LIN {X 0,Y 573.231,Z 369.083,A -85,B 0,C 180,E1 -2362.338,E2 -2362.338} C_VEL
LIN {X 0,Y 573.243,Z 369.081,A -85,B 0,C 180,E1 -2364.395,E2 -2364.395} C_VEL
LIN {X 0,Y 572.617,Z 369.161,A -85,B 0,C 180,E1 -2364.981,E2 -2364.981} C_VEL
LIN {X 0,Y 569.781,Z 369.515,A -85,B 0,C 180,E1 -2365.933,E2 -2365.933} C_VEL
LIN {X 0,Y 567.354,Z 369.816,A -85,B 0,C 180,E1 -2366.699,E2 -2366.699} C_VEL
LIN {X 0,Y 566.301,Z 369.946,A -85,B 0,C 180,E1 -2367.29,E2 -2367.29} C_VEL
LIN {X 0,Y 566.212,Z 369.956,A -85,B 0,C 180,E1 -2367.49,E2 -2367.49} C_VEL
LIN {X 0,Y 566.181,Z 369.961,A -85,B 0,C 180,E1 -2370.593,E2 -2370.593} C_VEL
LIN {X 0,Y 566.223,Z 369.955,A -85,B 0,C 180,E1 -2373.102,E2 -2373.102} C_VEL
LIN {X 0,Y 566.208,Z 369.958,A -85,B 0,C 180,E1 -2375.689,E2 -2375.689} C_VEL
LIN {X 0,Y 566.212,Z 369.957,A -85,B 0,C 180,E1 -2378.56,E2 -2378.56} C_VEL
LIN {X 0,Y 566.207,Z 369.958,A -85,B 0,C 180,E1 -2381.137,E2 -2381.137} C_VEL
LIN {X 0,Y 566.193,Z 369.96,A -85,B 0,C 180,E1 -2384.037,E2 -2384.037} C_VEL
LIN {X 0,Y 566.201,Z 369.96,A -85,B 0,C 180,E1 -2387.083,E2 -2387.083} C_VEL
LIN {X 0,Y 566.225,Z 369.955,A -85,B 0,C 180,E1 -2389.804,E2 -2389.804} C_VEL
LIN {X 0,Y 566.197,Z 369.96,A -85,B 0,C 180,E1 -2392.6,E2 -2392.6} C_VEL
LIN {X 0,Y 566.208,Z 369.957,A -85,B 0,C 180,E1 -2395.183,E2 -2395.183} C_VEL
LIN {X 0,Y 566.232,Z 369.955,A -85,B 0,C 180,E1 -2397.744,E2 -2397.744} C_VEL
LIN {X 0,Y 566.205,Z 369.959,A -85,B 0,C 180,E1 -2400.329,E2 -2400.329} C_VEL
LIN {X 0,Y 566.209,Z 369.958,A -85,B 0,C 180,E1 -2402.662,E2 -2402.662} C_VEL
LIN {X 0,Y 566.238,Z 369.953,A -85,B 0,C 180,E1 -2405.04,E2 -2405.04} C_VEL
LIN {X 0,Y 566.196,Z 369.96,A -85,B 0,C 180,E1 -2408.138,E2 -2408.138} C_VEL
LIN {X 0,Y 566.233,Z 369.954,A -85,B 0,C 180,E1 -2410.615,E2 -2410.615} C_VEL
LIN {X 0,Y 566.214,Z 369.958,A -85,B 0,C 180,E1 -2413.413,E2 -2413.413} C_VEL
LIN {X 0,Y 566.201,Z 369.958,A -85,B 0,C 180,E1 -2416.359,E2 -2416.359} C_VEL
LIN {X 0,Y 566.239,Z 369.953,A -85,B 0,C 180,E1 -2418.676,E2 -2418.676} C_VEL
LIN {X 0,Y 566.231,Z 369.956,A -85,B 0,C 180,E1 -2421.435,E2 -2421.435} C_VEL
LIN {X 0,Y 566.264,Z 369.951,A -85,B 0,C 180,E1 -2424.302,E2 -2424.302} C_VEL
LIN {X 0,Y 566.111,Z 369.972,A -85,B 0,C 180,E1 -2427.154,E2 -2427.154} C_VEL
LIN {X 0,Y 566.076,Z 369.978,A -85,B 0,C 180,E1 -2427.866,E2 -2427.866} C_VEL
LIN {X 0,Y 566.127,Z 372.153,A -85,B 0,C 180,E1 -2430,E2 -2430} C_VEL
LIN {X 0,Y 565.984,Z 374.62,A -85,B 0,C 180,E1 -2432.135,E2 -2432.135} C_VEL
LIN {X 0,Y 566.002,Z 377.796,A -85,B 0,C 180,E1 -2434.986,E2 -2434.986} C_VEL
LIN {X 0,Y 565.951,Z 381.039,A -85,B 0,C 180,E1 -2437.851,E2 -2437.851} C_VEL
LIN {X 0,Y 565.924,Z 384.456,A -85,B 0,C 180,E1 -2440.736,E2 -2440.736} C_VEL
LIN {X 0,Y 565.889,Z 388.157,A -85,B 0,C 180,E1 -2443.649,E2 -2443.649} C_VEL
LIN {X 0,Y 565.866,Z 391.969,A -85,B 0,C 180,E1 -2446.598,E2 -2446.598} C_VEL
LIN {X 0,Y 565.877,Z 395.756,A -85,B 0,C 180,E1 -2449.44,E2 -2449.44} C_VEL
LIN {X 0,Y 566.903,Z 403.162,A -85,B 0,C 180,E1 -2449.626,E2 -2449.626} C_VEL
LIN {X 0,Y 566.751,Z 416.361,A -85,B 0,C 180,E1 -2450.033,E2 -2450.033} C_VEL
LIN {X 0,Y 566.642,Z 427.451,A -85,B 0,C 180,E1 -2450.51,E2 -2450.51} C_VEL
LIN {X 0,Y 566.533,Z 439.685,A -85,B 0,C 180,E1 -2451.199,E2 -2451.199} C_VEL
LIN {X 0,Y 566.374,Z 450.264,A -85,B 0,C 180,E1 -2451.951,E2 -2451.951} C_VEL
LIN {X 0,Y 566.228,Z 460.09,A -85,B 0,C 180,E1 -2452.814,E2 -2452.814} C_VEL
LIN {X 0,Y 566.098,Z 469.138,A -85,B 0,C 180,E1 -2453.796,E2 -2453.796} C_VEL
LIN {X 0,Y 566.022,Z 476.522,A -85,B 0,C 180,E1 -2454.775,E2 -2454.775} C_VEL
LIN {X 0,Y 565.988,Z 483.713,A -85,B 0,C 180,E1 -2455.957,E2 -2455.957} C_VEL
LIN {X 0,Y 565.936,Z 488.503,A -85,B 0,C 180,E1 -2456.953,E2 -2456.953} C_VEL
LIN {X 0,Y 565.881,Z 492.991,A -85,B 0,C 180,E1 -2458.16,E2 -2458.16} C_VEL
LIN {X 0,Y 565.892,Z 495.248,A -85,B 0,C 180,E1 -2458.97,E2 -2458.97} C_VEL
LIN {X 0,Y 565.871,Z 497.003,A -85,B 0,C 180,E1 -2459.787,E2 -2459.787} C_VEL
LIN {X 0,Y 565.867,Z 498.577,A -85,B 0,C 180,E1 -2461.021,E2 -2461.021} C_VEL
LIN {X 0,Y 565.845,Z 498.934,A -85,B 0,C 180,E1 -2462.372,E2 -2462.372} C_VEL
LIN {X 0,Y 565.868,Z 497.946,A -85,B 0,C 180,E1 -2463.681,E2 -2463.681} C_VEL
LIN {X 0,Y 565.862,Z 495.687,A -85,B 0,C 180,E1 -2464.943,E2 -2464.943} C_VEL
LIN {X 0,Y 565.919,Z 492.176,A -85,B 0,C 180,E1 -2466.174,E2 -2466.174} C_VEL
LIN {X 0,Y 565.941,Z 486.955,A -85,B 0,C 180,E1 -2467.48,E2 -2467.48} C_VEL
LIN {X 0,Y 565.989,Z 480.61,A -85,B 0,C 180,E1 -2468.68,E2 -2468.68} C_VEL
LIN {X 0,Y 566.069,Z 474.047,A -85,B 0,C 180,E1 -2469.667,E2 -2469.667} C_VEL
LIN {X 0,Y 566.161,Z 464.892,A -85,B 0,C 180,E1 -2470.78,E2 -2470.78} C_VEL
LIN {X 0,Y 566.284,Z 455.077,A -85,B 0,C 180,E1 -2471.74,E2 -2471.74} C_VEL
LIN {X 0,Y 566.397,Z 444.775,A -85,B 0,C 180,E1 -2472.55,E2 -2472.55} C_VEL
LIN {X 0,Y 566.531,Z 433.437,A -85,B 0,C 180,E1 -2473.266,E2 -2473.266} C_VEL
LIN {X 0,Y 566.667,Z 421.184,A -85,B 0,C 180,E1 -2473.866,E2 -2473.866} C_VEL
LIN {X 0,Y 566.849,Z 408.099,A -85,B 0,C 180,E1 -2474.33,E2 -2474.33} C_VEL
LIN {X 0,Y 566.734,Z 401.219,A -85,B 0,C 180,E1 -2474.516,E2 -2474.516} C_VEL
LIN {X 0,Y 565.817,Z 395.661,A -85,B 0,C 180,E1 -2474.675,E2 -2474.675} C_VEL
LIN {X 0,Y 565.838,Z 391.468,A -85,B 0,C 180,E1 -2477.878,E2 -2477.878} C_VEL
LIN {X 0,Y 565.82,Z 387.838,A -85,B 0,C 180,E1 -2480.693,E2 -2480.693} C_VEL
LIN {X 0,Y 565.874,Z 383.867,A -85,B 0,C 180,E1 -2483.83,E2 -2483.83} C_VEL
LIN {X 0,Y 565.898,Z 381.098,A -85,B 0,C 180,E1 -2486.312,E2 -2486.312} C_VEL
LIN {X 0,Y 566,Z 378.247,A -85,B 0,C 180,E1 -2488.954,E2 -2488.954} C_VEL
LIN {X 0,Y 565.998,Z 374.957,A -85,B 0,C 180,E1 -2491.846,E2 -2491.846} C_VEL
LIN {X 0,Y 566.029,Z 372.197,A -85,B 0,C 180,E1 -2494.242,E2 -2494.242} C_VEL
LIN {X 0,Y 566.046,Z 370.404,A -85,B 0,C 180,E1 -2495.812,E2 -2495.812} C_VEL
LIN {X 0,Y 566.111,Z 369.973,A -85,B 0,C 180,E1 -2496.731,E2 -2496.731} C_VEL
LIN {X 0,Y 566.212,Z 369.957,A -85,B 0,C 180,E1 -2498.902,E2 -2498.902} C_VEL
LIN {X 0,Y 566.208,Z 369.958,A -85,B 0,C 180,E1 -2501.172,E2 -2501.172} C_VEL
LIN {X 0,Y 566.209,Z 369.96,A -85,B 0,C 180,E1 -2503.412,E2 -2503.412} C_VEL
LIN {X 0,Y 566.191,Z 369.959,A -85,B 0,C 180,E1 -2506.359,E2 -2506.359} C_VEL
LIN {X 0,Y 566.269,Z 369.949,A -85,B 0,C 180,E1 -2508.654,E2 -2508.654} C_VEL
LIN {X 0,Y 566.229,Z 369.954,A -85,B 0,C 180,E1 -2511.434,E2 -2511.434} C_VEL
LIN {X 0,Y 566.254,Z 369.954,A -85,B 0,C 180,E1 -2514.302,E2 -2514.302} C_VEL
LIN {X 0,Y 566.277,Z 369.951,A -85,B 0,C 180,E1 -2517.866,E2 -2517.866} C_VEL
LIN {X 0,Y 566.301,Z 369.945,A -85,B 0,C 180,E1 -2520.711,E2 -2520.711} C_VEL
LIN {X 0,Y 566.185,Z 369.96,A -85,B 0,C 180,E1 -2523.558,E2 -2523.558} C_VEL
LIN {X 0,Y 566.253,Z 369.951,A -85,B 0,C 180,E1 -2525.698,E2 -2525.698} C_VEL
LIN {X 0,Y 566.225,Z 369.955,A -85,B 0,C 180,E1 -2528.566,E2 -2528.566} C_VEL
LIN {X 0,Y 566.245,Z 369.953,A -85,B 0,C 180,E1 -2531.454,E2 -2531.454} C_VEL
LIN {X 0,Y 566.227,Z 369.954,A -85,B 0,C 180,E1 -2534.507,E2 -2534.507} C_VEL
LIN {X 0,Y 566.199,Z 369.961,A -85,B 0,C 180,E1 -2537.332,E2 -2537.332} C_VEL
LIN {X 0,Y 566.208,Z 369.956,A -85,B 0,C 180,E1 -2540.337,E2 -2540.337} C_VEL
LIN {X 0,Y 566.183,Z 369.963,A -85,B 0,C 180,E1 -2543.404,E2 -2543.404} C_VEL
LIN {X 0,Y 566.221,Z 369.959,A -85,B 0,C 180,E1 -2545.749,E2 -2545.749} C_VEL
LIN {X 0,Y 566.202,Z 369.961,A -85,B 0,C 180,E1 -2548.203,E2 -2548.203} C_VEL
LIN {X 0,Y 566.185,Z 369.96,A -85,B 0,C 180,E1 -2551.077,E2 -2551.077} C_VEL
LIN {X 0,Y 566.193,Z 369.959,A -85,B 0,C 180,E1 -2553.732,E2 -2553.732} C_VEL
LIN {X 0,Y 566.195,Z 369.962,A -85,B 0,C 180,E1 -2556.57,E2 -2556.57} C_VEL
LIN {X 0,Y 566.219,Z 369.958,A -85,B 0,C 180,E1 -2559.273,E2 -2559.273} C_VEL
LIN {X 0,Y 566.21,Z 369.956,A -85,B 0,C 180,E1 -2562.088,E2 -2562.088} C_VEL
LIN {X 0,Y 566.171,Z 369.964,A -85,B 0,C 180,E1 -2565.036,E2 -2565.036} C_VEL
LIN {X 0,Y 566.216,Z 369.957,A -85,B 0,C 180,E1 -2568.136,E2 -2568.136} C_VEL
LIN {X 0,Y 566.219,Z 369.957,A -85,B 0,C 180,E1 -2570.727,E2 -2570.727} C_VEL
LIN {X 0,Y 566.235,Z 369.971,A -85,B 0,C 180,E1 -2572.989,E2 -2572.989} C_VEL
LIN {X 0,Y 566.844,Z 373.918,A -85,B 0,C 180,E1 -2574.358,E2 -2574.358} C_VEL
LIN {X 0,Y 566.738,Z 381.862,A -85,B 0,C 180,E1 -2576.932,E2 -2576.932} C_VEL
LIN {X 0,Y 566.609,Z 389.805,A -85,B 0,C 180,E1 -2579.433,E2 -2579.433} C_VEL
LIN {X 0,Y 566.49,Z 399.072,A -85,B 0,C 180,E1 -2582.275,E2 -2582.275} C_VEL
LIN {X 0,Y 566.408,Z 408.339,A -85,B 0,C 180,E1 -2585.047,E2 -2585.047} C_VEL
LIN {X 0,Y 566.323,Z 418.93,A -85,B 0,C 180,E1 -2588.143,E2 -2588.143} C_VEL
LIN {X 0,Y 566.193,Z 429.521,A -85,B 0,C 180,E1 -2591.172,E2 -2591.172} C_VEL
LIN {X 0,Y 566.115,Z 440.112,A -85,B 0,C 180,E1 -2594.15,E2 -2594.15} C_VEL
LIN {X 0,Y 566.005,Z 450.703,A -85,B 0,C 180,E1 -2597.085,E2 -2597.085} C_VEL
LIN {X 0,Y 566.014,Z 451.53,A -85,B 0,C 180,E1 -2597.313,E2 -2597.313} C_VEL
LIN {X 0,Y 566.932,Z 458.375,A -85,B 0,C 180,E1 -2597.471,E2 -2597.471} C_VEL
LIN {X 0,Y 566.842,Z 470.499,A -85,B 0,C 180,E1 -2597.787,E2 -2597.787} C_VEL
LIN {X 0,Y 566.679,Z 482.321,A -85,B 0,C 180,E1 -2598.228,E2 -2598.228} C_VEL
LIN {X 0,Y 566.54,Z 494.84,A -85,B 0,C 180,E1 -2598.86,E2 -2598.86} C_VEL
LIN {X 0,Y 566.433,Z 505.479,A -85,B 0,C 180,E1 -2599.545,E2 -2599.545} C_VEL
LIN {X 0,Y 566.301,Z 515.647,A -85,B 0,C 180,E1 -2600.355,E2 -2600.355} C_VEL
LIN {X 0,Y 566.166,Z 524.787,A -85,B 0,C 180,E1 -2601.253,E2 -2601.253} C_VEL
LIN {X 0,Y 566.08,Z 533.69,A -85,B 0,C 180,E1 -2602.33,E2 -2602.33} C_VEL
LIN {X 0,Y 565.967,Z 540.955,A -85,B 0,C 180,E1 -2603.422,E2 -2603.422} C_VEL
LIN {X 0,Y 566.004,Z 545.68,A -85,B 0,C 180,E1 -2604.299,E2 -2604.299} C_VEL
LIN {X 0,Y 565.933,Z 550.371,A -85,B 0,C 180,E1 -2605.37,E2 -2605.37} C_VEL
LIN {X 0,Y 565.927,Z 553.956,A -85,B 0,C 180,E1 -2606.44,E2 -2606.44} C_VEL
LIN {X 0,Y 565.878,Z 555.808,A -85,B 0,C 180,E1 -2607.152,E2 -2607.152} C_VEL
LIN {X 0,Y 565.84,Z 557.2,A -85,B 0,C 180,E1 -2607.864,E2 -2607.864} C_VEL
LIN {X 0,Y 565.841,Z 558.784,A -85,B 0,C 180,E1 -2609.288,E2 -2609.288} C_VEL
LIN {X 0,Y 565.839,Z 559,A -85,B 0,C 180,E1 -2610,E2 -2610} C_VEL
LIN {X 0,Y 565.846,Z 558.186,A -85,B 0,C 180,E1 -2611.423,E2 -2611.423} C_VEL
LIN {X 0,Y 565.84,Z 557.201,A -85,B 0,C 180,E1 -2612.135,E2 -2612.135} C_VEL
LIN {X 0,Y 565.878,Z 555.81,A -85,B 0,C 180,E1 -2612.847,E2 -2612.847} C_VEL
LIN {X 0,Y 565.926,Z 552.897,A -85,B 0,C 180,E1 -2613.916,E2 -2613.916} C_VEL
LIN {X 0,Y 565.878,Z 548.951,A -85,B 0,C 180,E1 -2614.987,E2 -2614.987} C_VEL
LIN {X 0,Y 566.002,Z 543.868,A -85,B 0,C 180,E1 -2616.058,E2 -2616.058} C_VEL
LIN {X 0,Y 566.04,Z 537.472,A -85,B 0,C 180,E1 -2617.132,E2 -2617.132} C_VEL
LIN {X 0,Y 566.133,Z 529.481,A -85,B 0,C 180,E1 -2618.207,E2 -2618.207} C_VEL
LIN {X 0,Y 566.229,Z 521.34,A -85,B 0,C 180,E1 -2619.105,E2 -2619.105} C_VEL
LIN {X 0,Y 566.346,Z 511.407,A -85,B 0,C 180,E1 -2620.004,E2 -2620.004} C_VEL
LIN {X 0,Y 566.522,Z 500.32,A -85,B 0,C 180,E1 -2620.805,E2 -2620.805} C_VEL
LIN {X 0,Y 566.607,Z 487.959,A -85,B 0,C 180,E1 -2621.509,E2 -2621.509} C_VEL
LIN {X 0,Y 566.771,Z 475.779,A -85,B 0,C 180,E1 -2622.033,E2 -2622.033} C_VEL
LIN {X 0,Y 566.915,Z 463.282,A -85,B 0,C 180,E1 -2622.416,E2 -2622.416} C_VEL
LIN {X 0,Y 566.732,Z 456.109,A -85,B 0,C 180,E1 -2622.579,E2 -2622.579} C_VEL
LIN {X 0,Y 566.014,Z 451.532,A -85,B 0,C 180,E1 -2622.686,E2 -2622.686} C_VEL
LIN {X 0,Y 566.088,Z 441.437,A -85,B 0,C 180,E1 -2625.481,E2 -2625.481} C_VEL
LIN {X 0,Y 566.174,Z 430.846,A -85,B 0,C 180,E1 -2628.453,E2 -2628.453} C_VEL
LIN {X 0,Y 566.238,Z 421.579,A -85,B 0,C 180,E1 -2631.096,E2 -2631.096} C_VEL
LIN {X 0,Y 566.341,Z 412.312,A -85,B 0,C 180,E1 -2633.784,E2 -2633.784} C_VEL
LIN {X 0,Y 566.477,Z 403.045,A -85,B 0,C 180,E1 -2636.527,E2 -2636.527} C_VEL
LIN {X 0,Y 566.539,Z 393.778,A -85,B 0,C 180,E1 -2639.34,E2 -2639.34} C_VEL
LIN {X 0,Y 566.75,Z 384.511,A -85,B 0,C 180,E1 -2642.223,E2 -2642.223} C_VEL
LIN {X 0,Y 566.836,Z 376.568,A -85,B 0,C 180,E1 -2644.773,E2 -2644.773} C_VEL
LIN {X 0,Y 566.619,Z 372.042,A -85,B 0,C 180,E1 -2646.271,E2 -2646.271} C_VEL
LIN {X 0,Y 566.234,Z 369.955,A -85,B 0,C 180,E1 -2647.01,E2 -2647.01} C_VEL
LIN {X 0,Y 566.212,Z 369.959,A -85,B 0,C 180,E1 -2649.685,E2 -2649.685} C_VEL
LIN {X 0,Y 566.21,Z 369.958,A -85,B 0,C 180,E1 -2652.086,E2 -2652.086} C_VEL
LIN {X 0,Y 566.169,Z 369.965,A -85,B 0,C 180,E1 -2655.035,E2 -2655.035} C_VEL
LIN {X 0,Y 566.212,Z 369.957,A -85,B 0,C 180,E1 -2658.135,E2 -2658.135} C_VEL
LIN {X 0,Y 566.216,Z 369.959,A -85,B 0,C 180,E1 -2660.726,E2 -2660.726} C_VEL
LIN {X 0,Y 566.212,Z 369.958,A -85,B 0,C 180,E1 -2663.783,E2 -2663.783} C_VEL
LIN {X 0,Y 566.223,Z 369.958,A -85,B 0,C 180,E1 -2666.262,E2 -2666.262} C_VEL
LIN {X 0,Y 566.192,Z 369.959,A -85,B 0,C 180,E1 -2668.921,E2 -2668.921} C_VEL
LIN {X 0,Y 566.22,Z 369.957,A -85,B 0,C 180,E1 -2671.858,E2 -2671.858} C_VEL
LIN {X 0,Y 566.216,Z 369.957,A -85,B 0,C 180,E1 -2674.251,E2 -2674.251} C_VEL
LIN {X 0,Y 566.183,Z 369.96,A -85,B 0,C 180,E1 -2676.713,E2 -2676.713} C_VEL
LIN {X 0,Y 566.212,Z 369.957,A -85,B 0,C 180,E1 -2679.663,E2 -2679.663} C_VEL
LIN {X 0,Y 566.197,Z 369.96,A -85,B 0,C 180,E1 -2682.668,E2 -2682.668} C_VEL
LIN {X 0,Y 566.224,Z 369.955,A -85,B 0,C 180,E1 -2685.627,E2 -2685.627} C_VEL
LIN {X 0,Y 566.266,Z 369.951,A -85,B 0,C 180,E1 -2688.654,E2 -2688.654} C_VEL
LIN {X 0,Y 566.24,Z 369.955,A -85,B 0,C 180,E1 -2691.435,E2 -2691.435} C_VEL
LIN {X 0,Y 566.25,Z 369.952,A -85,B 0,C 180,E1 -2694.302,E2 -2694.302} C_VEL
LIN {X 0,Y 566.272,Z 369.949,A -85,B 0,C 180,E1 -2697.866,E2 -2697.866} C_VEL
LIN {X 0,Y 566.302,Z 369.947,A -85,B 0,C 180,E1 -2700.711,E2 -2700.711} C_VEL
LIN {X 0,Y 566.27,Z 369.951,A -85,B 0,C 180,E1 -2702.846,E2 -2702.846} C_VEL
LIN {X 0,Y 566.254,Z 369.951,A -85,B 0,C 180,E1 -2705.698,E2 -2705.698} C_VEL
LIN {X 0,Y 566.241,Z 369.954,A -85,B 0,C 180,E1 -2708.566,E2 -2708.566} C_VEL
LIN {X 0,Y 566.242,Z 369.955,A -85,B 0,C 180,E1 -2711.454,E2 -2711.454} C_VEL
LIN {X 0,Y 566.225,Z 369.956,A -85,B 0,C 180,E1 -2714.507,E2 -2714.507} C_VEL
LIN {X 0,Y 566.195,Z 369.959,A -85,B 0,C 180,E1 -2717.332,E2 -2717.332} C_VEL
LIN {X 0,Y 566.213,Z 369.959,A -85,B 0,C 180,E1 -2720.337,E2 -2720.337} C_VEL
LIN {X 0,Y 566.182,Z 369.96,A -85,B 0,C 180,E1 -2723.404,E2 -2723.404} C_VEL
LIN {X 0,Y 566.217,Z 369.957,A -85,B 0,C 180,E1 -2725.749,E2 -2725.749} C_VEL
LIN {X 0,Y 566.212,Z 369.956,A -85,B 0,C 180,E1 -2727.49,E2 -2727.49} C_VEL
LIN {X 0,Y 565.531,Z 370.044,A -85,B 0,C 180,E1 -2728.084,E2 -2728.084} C_VEL
LIN {X 0,Y 562.659,Z 370.4,A -85,B 0,C 180,E1 -2729.048,E2 -2729.048} C_VEL
LIN {X 0,Y 560.245,Z 370.7,A -85,B 0,C 180,E1 -2729.823,E2 -2729.823} C_VEL
LIN {X 0,Y 559.218,Z 370.83,A -85,B 0,C 180,E1 -2730.422,E2 -2730.422} C_VEL
LIN {X 0,Y 559.138,Z 370.836,A -85,B 0,C 180,E1 -2730.624,E2 -2730.624} C_VEL
LIN {X 0,Y 559.172,Z 370.835,A -85,B 0,C 180,E1 -2733.575,E2 -2733.575} C_VEL
LIN {X 0,Y 559.185,Z 370.832,A -85,B 0,C 180,E1 -2736.452,E2 -2736.452} C_VEL
LIN {X 0,Y 559.174,Z 370.834,A -85,B 0,C 180,E1 -2738.934,E2 -2738.934} C_VEL
LIN {X 0,Y 559.187,Z 370.832,A -85,B 0,C 180,E1 -2741.768,E2 -2741.768} C_VEL
LIN {X 0,Y 559.135,Z 370.84,A -85,B 0,C 180,E1 -2744.74,E2 -2744.74} C_VEL
LIN {X 0,Y 559.174,Z 370.834,A -85,B 0,C 180,E1 -2747.863,E2 -2747.863} C_VEL
LIN {X 0,Y 559.183,Z 370.834,A -85,B 0,C 180,E1 -2750.136,E2 -2750.136} C_VEL
LIN {X 0,Y 559.143,Z 370.837,A -85,B 0,C 180,E1 -2752.893,E2 -2752.893} C_VEL
LIN {X 0,Y 559.165,Z 370.836,A -85,B 0,C 180,E1 -2756.052,E2 -2756.052} C_VEL
LIN {X 0,Y 559.163,Z 370.836,A -85,B 0,C 180,E1 -2758.982,E2 -2758.982} C_VEL
LIN {X 0,Y 559.169,Z 370.835,A -85,B 0,C 180,E1 -2761.62,E2 -2761.62} C_VEL
LIN {X 0,Y 559.184,Z 370.833,A -85,B 0,C 180,E1 -2763.904,E2 -2763.904} C_VEL
LIN {X 0,Y 559.159,Z 370.836,A -85,B 0,C 180,E1 -2766.568,E2 -2766.568} C_VEL
LIN {X 0,Y 559.177,Z 370.834,A -85,B 0,C 180,E1 -2769.396,E2 -2769.396} C_VEL
LIN {X 0,Y 559.144,Z 370.838,A -85,B 0,C 180,E1 -2771.686,E2 -2771.686} C_VEL
LIN {X 0,Y 559.166,Z 370.835,A -85,B 0,C 180,E1 -2773.948,E2 -2773.948} C_VEL
LIN {X 0,Y 559.176,Z 370.833,A -85,B 0,C 180,E1 -2776.185,E2 -2776.185} C_VEL
LIN {X 0,Y 559.199,Z 370.833,A -85,B 0,C 180,E1 -2779.134,E2 -2779.134} C_VEL
LIN {X 0,Y 559.204,Z 370.83,A -85,B 0,C 180,E1 -2782.054,E2 -2782.054} C_VEL
LIN {X 0,Y 559.254,Z 370.823,A -85,B 0,C 180,E1 -2784.954,E2 -2784.954} C_VEL
LIN {X 0,Y 559.042,Z 370.854,A -85,B 0,C 180,E1 -2787.839,E2 -2787.839} C_VEL
LIN {X 0,Y 559.027,Z 371.145,A -85,B 0,C 180,E1 -2788.559,E2 -2788.559} C_VEL
LIN {X 0,Y 559.008,Z 373.635,A -85,B 0,C 180,E1 -2790.721,E2 -2790.721} C_VEL
LIN {X 0,Y 558.909,Z 376.925,A -85,B 0,C 180,E1 -2793.605,E2 -2793.605} C_VEL
LIN {X 0,Y 558.901,Z 379.335,A -85,B 0,C 180,E1 -2795.774,E2 -2795.774} C_VEL
LIN {X 0,Y 558.871,Z 382.614,A -85,B 0,C 180,E1 -2798.679,E2 -2798.679} C_VEL
LIN {X 0,Y 558.834,Z 385.979,A -85,B 0,C 180,E1 -2801.608,E2 -2801.608} C_VEL
LIN {X 0,Y 558.809,Z 389.63,A -85,B 0,C 180,E1 -2804.568,E2 -2804.568} C_VEL
LIN {X 0,Y 558.751,Z 393.48,A -85,B 0,C 180,E1 -2807.57,E2 -2807.57} C_VEL
LIN {X 0,Y 558.771,Z 395.776,A -85,B 0,C 180,E1 -2809.277,E2 -2809.277} C_VEL
LIN {X 0,Y 559.969,Z 403.84,A -85,B 0,C 180,E1 -2809.487,E2 -2809.487} C_VEL
LIN {X 0,Y 559.836,Z 415.759,A -85,B 0,C 180,E1 -2809.86,E2 -2809.86} C_VEL
LIN {X 0,Y 559.658,Z 428.016,A -85,B 0,C 180,E1 -2810.394,E2 -2810.394} C_VEL
LIN {X 0,Y 559.54,Z 439.834,A -85,B 0,C 180,E1 -2811.072,E2 -2811.072} C_VEL
LIN {X 0,Y 559.36,Z 450.423,A -85,B 0,C 180,E1 -2811.835,E2 -2811.835} C_VEL
LIN {X 0,Y 559.205,Z 460.456,A -85,B 0,C 180,E1 -2812.734,E2 -2812.734} C_VEL
LIN {X 0,Y 559.036,Z 469.387,A -85,B 0,C 180,E1 -2813.721,E2 -2813.721} C_VEL
LIN {X 0,Y 558.966,Z 477.487,A -85,B 0,C 180,E1 -2814.825,E2 -2814.825} C_VEL
LIN {X 0,Y 558.909,Z 483.87,A -85,B 0,C 180,E1 -2815.91,E2 -2815.91} C_VEL
LIN {X 0,Y 558.848,Z 488.636,A -85,B 0,C 180,E1 -2816.919,E2 -2816.919} C_VEL
LIN {X 0,Y 558.792,Z 493.576,A -85,B 0,C 180,E1 -2818.309,E2 -2818.309} C_VEL
LIN {X 0,Y 558.772,Z 497.053,A -85,B 0,C 180,E1 -2819.789,E2 -2819.789} C_VEL
LIN {X 0,Y 558.763,Z 498.71,A -85,B 0,C 180,E1 -2821.208,E2 -2821.208} C_VEL
LIN {X 0,Y 558.76,Z 498.89,A -85,B 0,C 180,E1 -2822.571,E2 -2822.571} C_VEL
LIN {X 0,Y 558.771,Z 497.69,A -85,B 0,C 180,E1 -2823.888,E2 -2823.888} C_VEL
LIN {X 0,Y 558.782,Z 495.241,A -85,B 0,C 180,E1 -2825.161,E2 -2825.161} C_VEL
LIN {X 0,Y 558.814,Z 491.588,A -85,B 0,C 180,E1 -2826.399,E2 -2826.399} C_VEL
LIN {X 0,Y 558.875,Z 486.709,A -85,B 0,C 180,E1 -2827.604,E2 -2827.604} C_VEL
LIN {X 0,Y 558.907,Z 480.552,A -85,B 0,C 180,E1 -2828.774,E2 -2828.774} C_VEL
LIN {X 0,Y 559.023,Z 472.853,A -85,B 0,C 180,E1 -2829.924,E2 -2829.924} C_VEL
LIN {X 0,Y 559.112,Z 464.514,A -85,B 0,C 180,E1 -2830.933,E2 -2830.933} C_VEL
LIN {X 0,Y 559.271,Z 455.125,A -85,B 0,C 180,E1 -2831.859,E2 -2831.859} C_VEL
LIN {X 0,Y 559.411,Z 444.27,A -85,B 0,C 180,E1 -2832.719,E2 -2832.719} C_VEL
LIN {X 0,Y 559.54,Z 432.266,A -85,B 0,C 180,E1 -2833.475,E2 -2833.475} C_VEL
LIN {X 0,Y 559.729,Z 420.751,A -85,B 0,C 180,E1 -2834.032,E2 -2834.032} C_VEL
LIN {X 0,Y 559.895,Z 407.507,A -85,B 0,C 180,E1 -2834.503,E2 -2834.503} C_VEL
LIN {X 0,Y 559.707,Z 401.571,A -85,B 0,C 180,E1 -2834.666,E2 -2834.666} C_VEL
LIN {X 0,Y 558.722,Z 395.672,A -85,B 0,C 180,E1 -2834.83,E2 -2834.83} C_VEL
LIN {X 0,Y 558.742,Z 391.69,A -85,B 0,C 180,E1 -2837.911,E2 -2837.911} C_VEL
LIN {X 0,Y 558.76,Z 388.889,A -85,B 0,C 180,E1 -2840.106,E2 -2840.106} C_VEL
LIN {X 0,Y 558.756,Z 385.618,A -85,B 0,C 180,E1 -2842.861,E2 -2842.861} C_VEL
LIN {X 0,Y 558.832,Z 382.587,A -85,B 0,C 180,E1 -2845.533,E2 -2845.533} C_VEL
LIN {X 0,Y 558.898,Z 379.772,A -85,B 0,C 180,E1 -2848.12,E2 -2848.12} C_VEL
LIN {X 0,Y 558.925,Z 376.983,A -85,B 0,C 180,E1 -2850.633,E2 -2850.633} C_VEL
LIN {X 0,Y 558.935,Z 374.024,A -85,B 0,C 180,E1 -2853.219,E2 -2853.219} C_VEL
LIN {X 0,Y 558.979,Z 371.475,A -85,B 0,C 180,E1 -2855.486,E2 -2855.486} C_VEL
LIN {X 0,Y 559.052,Z 370.852,A -85,B 0,C 180,E1 -2856.59,E2 -2856.59} C_VEL
LIN {X 0,Y 559.181,Z 370.833,A -85,B 0,C 180,E1 -2859.395,E2 -2859.395} C_VEL
LIN {X 0,Y 559.149,Z 370.836,A -85,B 0,C 180,E1 -2861.686,E2 -2861.686} C_VEL
LIN {X 0,Y 559.161,Z 370.834,A -85,B 0,C 180,E1 -2863.948,E2 -2863.948} C_VEL
LIN {X 0,Y 559.165,Z 370.834,A -85,B 0,C 180,E1 -2866.184,E2 -2866.184} C_VEL
LIN {X 0,Y 559.203,Z 370.83,A -85,B 0,C 180,E1 -2869.134,E2 -2869.134} C_VEL
LIN {X 0,Y 559.199,Z 370.831,A -85,B 0,C 180,E1 -2872.053,E2 -2872.053} C_VEL
LIN {X 0,Y 559.254,Z 370.822,A -85,B 0,C 180,E1 -2874.953,E2 -2874.953} C_VEL
LIN {X 0,Y 559.248,Z 370.826,A -85,B 0,C 180,E1 -2877.839,E2 -2877.839} C_VEL
LIN {X 0,Y 559.271,Z 370.821,A -85,B 0,C 180,E1 -2880.72,E2 -2880.72} C_VEL
LIN {X 0,Y 559.235,Z 370.827,A -85,B 0,C 180,E1 -2882.881,E2 -2882.881} C_VEL
LIN {X 0,Y 559.222,Z 370.827,A -85,B 0,C 180,E1 -2885.77,E2 -2885.77} C_VEL
LIN {X 0,Y 559.184,Z 370.833,A -85,B 0,C 180,E1 -2888.674,E2 -2888.674} C_VEL
LIN {X 0,Y 559.203,Z 370.83,A -85,B 0,C 180,E1 -2891.6,E2 -2891.6} C_VEL
LIN {X 0,Y 559.193,Z 370.831,A -85,B 0,C 180,E1 -2894.596,E2 -2894.596} C_VEL
LIN {X 0,Y 559.158,Z 370.836,A -85,B 0,C 180,E1 -2897.557,E2 -2897.557} C_VEL
LIN {X 0,Y 559.166,Z 370.836,A -85,B 0,C 180,E1 -2899.838,E2 -2899.838} C_VEL
LIN {X 0,Y 559.136,Z 370.841,A -85,B 0,C 180,E1 -2902.153,E2 -2902.153} C_VEL
LIN {X 0,Y 559.174,Z 370.833,A -85,B 0,C 180,E1 -2905.188,E2 -2905.188} C_VEL
LIN {X 0,Y 559.19,Z 370.831,A -85,B 0,C 180,E1 -2907.712,E2 -2907.712} C_VEL
LIN {X 0,Y 559.148,Z 370.837,A -85,B 0,C 180,E1 -2910.183,E2 -2910.183} C_VEL
LIN {X 0,Y 559.148,Z 370.837,A -85,B 0,C 180,E1 -2912.716,E2 -2912.716} C_VEL
LIN {X 0,Y 559.125,Z 370.842,A -85,B 0,C 180,E1 -2915.324,E2 -2915.324} C_VEL
LIN {X 0,Y 559.132,Z 370.841,A -85,B 0,C 180,E1 -2918.018,E2 -2918.018} C_VEL
LIN {X 0,Y 559.174,Z 370.833,A -85,B 0,C 180,E1 -2920.811,E2 -2920.811} C_VEL
LIN {X 0,Y 559.138,Z 370.839,A -85,B 0,C 180,E1 -2923.734,E2 -2923.734} C_VEL
LIN {X 0,Y 559.144,Z 370.838,A -85,B 0,C 180,E1 -2926.804,E2 -2926.804} C_VEL
LIN {X 0,Y 559.175,Z 370.835,A -85,B 0,C 180,E1 -2929.19,E2 -2929.19} C_VEL
LIN {X 0,Y 559.131,Z 370.84,A -85,B 0,C 180,E1 -2931.983,E2 -2931.983} C_VEL
LIN {X 0,Y 559.212,Z 371.017,A -85,B 0,C 180,E1 -2932.8,E2 -2932.8} C_VEL
LIN {X 0,Y 559.884,Z 375.26,A -85,B 0,C 180,E1 -2934.29,E2 -2934.29} C_VEL
LIN {X 0,Y 559.857,Z 381.862,A -85,B 0,C 180,E1 -2936.473,E2 -2936.473} C_VEL
LIN {X 0,Y 559.656,Z 389.805,A -85,B 0,C 180,E1 -2939.012,E2 -2939.012} C_VEL
LIN {X 0,Y 559.542,Z 399.159,A -85,B 0,C 180,E1 -2941.927,E2 -2941.927} C_VEL
LIN {X 0,Y 559.398,Z 408.516,A -85,B 0,C 180,E1 -2944.766,E2 -2944.766} C_VEL
LIN {X 0,Y 559.291,Z 418.93,A -85,B 0,C 180,E1 -2947.854,E2 -2947.854} C_VEL
LIN {X 0,Y 559.149,Z 429.521,A -85,B 0,C 180,E1 -2950.926,E2 -2950.926} C_VEL
LIN {X 0,Y 559.057,Z 438.788,A -85,B 0,C 180,E1 -2953.57,E2 -2953.57} C_VEL
LIN {X 0,Y 558.963,Z 449.379,A -85,B 0,C 180,E1 -2956.55,E2 -2956.55} C_VEL
LIN {X 0,Y 558.94,Z 451.53,A -85,B 0,C 180,E1 -2957.15,E2 -2957.15} C_VEL
LIN {X 0,Y 560.02,Z 459.514,A -85,B 0,C 180,E1 -2957.337,E2 -2957.337} C_VEL
LIN {X 0,Y 559.882,Z 471.879,A -85,B 0,C 180,E1 -2957.679,E2 -2957.679} C_VEL
LIN {X 0,Y 559.717,Z 484.284,A -85,B 0,C 180,E1 -2958.171,E2 -2958.171} C_VEL
LIN {X 0,Y 559.557,Z 495.668,A -85,B 0,C 180,E1 -2958.768,E2 -2958.768} C_VEL
LIN {X 0,Y 559.428,Z 506.747,A -85,B 0,C 180,E1 -2959.504,E2 -2959.504} C_VEL
LIN {X 0,Y 559.244,Z 517.601,A -85,B 0,C 180,E1 -2960.415,E2 -2960.415} C_VEL
LIN {X 0,Y 559.127,Z 526.413,A -85,B 0,C 180,E1 -2961.325,E2 -2961.325} C_VEL
LIN {X 0,Y 558.996,Z 535,A -85,B 0,C 180,E1 -2962.414,E2 -2962.414} C_VEL
LIN {X 0,Y 558.885,Z 542.688,A -85,B 0,C 180,E1 -2963.649,E2 -2963.649} C_VEL
LIN {X 0,Y 558.869,Z 547.365,A -85,B 0,C 180,E1 -2964.588,E2 -2964.588} C_VEL
LIN {X 0,Y 558.869,Z 551.677,A -85,B 0,C 180,E1 -2965.673,E2 -2965.673} C_VEL
LIN {X 0,Y 558.836,Z 553.956,A -85,B 0,C 180,E1 -2966.395,E2 -2966.395} C_VEL
LIN {X 0,Y 558.799,Z 555.808,A -85,B 0,C 180,E1 -2967.116,E2 -2967.116} C_VEL
LIN {X 0,Y 558.746,Z 557.199,A -85,B 0,C 180,E1 -2967.837,E2 -2967.837} C_VEL
LIN {X 0,Y 558.741,Z 558.784,A -85,B 0,C 180,E1 -2969.279,E2 -2969.279} C_VEL
LIN {X 0,Y 558.74,Z 559,A -85,B 0,C 180,E1 -2970,E2 -2970} C_VEL
LIN {X 0,Y 558.745,Z 558.186,A -85,B 0,C 180,E1 -2971.441,E2 -2971.441} C_VEL
LIN {X 0,Y 558.746,Z 557.201,A -85,B 0,C 180,E1 -2972.162,E2 -2972.162} C_VEL
LIN {X 0,Y 558.799,Z 555.81,A -85,B 0,C 180,E1 -2972.883,E2 -2972.883} C_VEL
LIN {X 0,Y 558.844,Z 552.897,A -85,B 0,C 180,E1 -2973.966,E2 -2973.966} C_VEL
LIN {X 0,Y 558.798,Z 548.95,A -85,B 0,C 180,E1 -2975.051,E2 -2975.051} C_VEL
LIN {X 0,Y 558.921,Z 543.868,A -85,B 0,C 180,E1 -2976.135,E2 -2976.135} C_VEL
LIN {X 0,Y 558.977,Z 537.472,A -85,B 0,C 180,E1 -2977.223,E2 -2977.223} C_VEL
LIN {X 0,Y 559.098,Z 529.481,A -85,B 0,C 180,E1 -2978.311,E2 -2978.311} C_VEL
LIN {X 0,Y 559.194,Z 521.34,A -85,B 0,C 180,E1 -2979.221,E2 -2979.221} C_VEL
LIN {X 0,Y 559.347,Z 511.407,A -85,B 0,C 180,E1 -2980.131,E2 -2980.131} C_VEL
LIN {X 0,Y 559.539,Z 500.416,A -85,B 0,C 180,E1 -2980.936,E2 -2980.936} C_VEL
LIN {X 0,Y 559.635,Z 488.831,A -85,B 0,C 180,E1 -2981.61,E2 -2981.61} C_VEL
LIN {X 0,Y 559.81,Z 476.999,A -85,B 0,C 180,E1 -2982.138,E2 -2982.138} C_VEL
LIN {X 0,Y 559.952,Z 464.195,A -85,B 0,C 180,E1 -2982.549,E2 -2982.549} C_VEL
LIN {X 0,Y 559.816,Z 456.967,A -85,B 0,C 180,E1 -2982.72,E2 -2982.72} C_VEL
LIN {X 0,Y 558.939,Z 451.532,A -85,B 0,C 180,E1 -2982.85,E2 -2982.85} C_VEL
LIN {X 0,Y 559.053,Z 441.437,A -85,B 0,C 180,E1 -2985.681,E2 -2985.681} C_VEL
LIN {X 0,Y 559.14,Z 430.846,A -85,B 0,C 180,E1 -2988.694,E2 -2988.694} C_VEL
LIN {X 0,Y 559.222,Z 420.92,A -85,B 0,C 180,E1 -2991.566,E2 -2991.566} C_VEL
LIN {X 0,Y 559.369,Z 410.988,A -85,B 0,C 180,E1 -2994.494,E2 -2994.494} C_VEL
LIN {X 0,Y 559.471,Z 401.721,A -85,B 0,C 180,E1 -2997.29,E2 -2997.29} C_VEL
LIN {X 0,Y 559.637,Z 392.454,A -85,B 0,C 180,E1 -3000.153,E2 -3000.153} C_VEL
LIN {X 0,Y 559.768,Z 384.329,A -85,B 0,C 180,E1 -3002.733,E2 -3002.733} C_VEL
LIN {X 0,Y 559.89,Z 376.376,A -85,B 0,C 180,E1 -3005.322,E2 -3005.322} C_VEL
LIN {X 0,Y 559.259,Z 371.193,A -85,B 0,C 180,E1 -3007.098,E2 -3007.098} C_VEL
LIN {X 0,Y 559.169,Z 370.837,A -85,B 0,C 180,E1 -3007.301,E2 -3007.301} C_VEL
LIN {X 0,Y 559.157,Z 370.836,A -85,B 0,C 180,E1 -3009.941,E2 -3009.941} C_VEL
LIN {X 0,Y 559.16,Z 370.837,A -85,B 0,C 180,E1 -3012.742,E2 -3012.742} C_VEL
LIN {X 0,Y 559.148,Z 370.837,A -85,B 0,C 180,E1 -3015.76,E2 -3015.76} C_VEL
LIN {X 0,Y 559.186,Z 370.833,A -85,B 0,C 180,E1 -3018.232,E2 -3018.232} C_VEL
LIN {X 0,Y 559.172,Z 370.834,A -85,B 0,C 180,E1 -3021.19,E2 -3021.19} C_VEL
LIN {X 0,Y 559.167,Z 370.836,A -85,B 0,C 180,E1 -3023.791,E2 -3023.791} C_VEL
LIN {X 0,Y 559.171,Z 370.835,A -85,B 0,C 180,E1 -3026.426,E2 -3026.426} C_VEL
LIN {X 0,Y 559.155,Z 370.836,A -85,B 0,C 180,E1 -3028.981,E2 -3028.981} C_VEL
LIN {X 0,Y 559.188,Z 370.831,A -85,B 0,C 180,E1 -3032.288,E2 -3032.288} C_VEL
LIN {X 0,Y 559.171,Z 370.835,A -85,B 0,C 180,E1 -3034.812,E2 -3034.812} C_VEL
LIN {X 0,Y 559.134,Z 370.837,A -85,B 0,C 180,E1 -3037.847,E2 -3037.847} C_VEL
LIN {X 0,Y 559.189,Z 370.833,A -85,B 0,C 180,E1 -3040.492,E2 -3040.492} C_VEL
LIN {X 0,Y 559.178,Z 370.833,A -85,B 0,C 180,E1 -3043.197,E2 -3043.197} C_VEL
LIN {X 0,Y 559.164,Z 370.837,A -85,B 0,C 180,E1 -3046.184,E2 -3046.184} C_VEL
LIN {X 0,Y 559.202,Z 370.831,A -85,B 0,C 180,E1 -3049.134,E2 -3049.134} C_VEL
LIN {X 0,Y 559.204,Z 370.83,A -85,B 0,C 180,E1 -3052.054,E2 -3052.054} C_VEL
LIN {X 0,Y 559.244,Z 370.827,A -85,B 0,C 180,E1 -3054.953,E2 -3054.953} C_VEL
LIN {X 0,Y 559.243,Z 370.824,A -85,B 0,C 180,E1 -3057.839,E2 -3057.839} C_VEL
LIN {X 0,Y 559.271,Z 370.822,A -85,B 0,C 180,E1 -3060.72,E2 -3060.72} C_VEL
LIN {X 0,Y 559.236,Z 370.827,A -85,B 0,C 180,E1 -3062.881,E2 -3062.881} C_VEL
LIN {X 0,Y 559.223,Z 370.827,A -85,B 0,C 180,E1 -3065.77,E2 -3065.77} C_VEL
LIN {X 0,Y 559.196,Z 370.831,A -85,B 0,C 180,E1 -3068.674,E2 -3068.674} C_VEL
LIN {X 0,Y 559.2,Z 370.832,A -85,B 0,C 180,E1 -3071.601,E2 -3071.601} C_VEL
LIN {X 0,Y 559.19,Z 370.832,A -85,B 0,C 180,E1 -3074.596,E2 -3074.596} C_VEL
LIN {X 0,Y 559.155,Z 370.835,A -85,B 0,C 180,E1 -3077.557,E2 -3077.557} C_VEL
LIN {X 0,Y 559.167,Z 370.834,A -85,B 0,C 180,E1 -3079.838,E2 -3079.838} C_VEL
LIN {X 0,Y 559.135,Z 370.838,A -85,B 0,C 180,E1 -3082.153,E2 -3082.153} C_VEL
LIN {X 0,Y 559.172,Z 370.833,A -85,B 0,C 180,E1 -3085.188,E2 -3085.188} C_VEL
LIN {X 0,Y 559.189,Z 370.831,A -85,B 0,C 180,E1 -3087.712,E2 -3087.712} C_VEL
LIN {X 0,Y 559.138,Z 370.836,A -85,B 0,C 180,E1 -3090.624,E2 -3090.624} C_VEL
LIN {X 0,Y 558.48,Z 370.921,A -85,B 0,C 180,E1 -3091.226,E2 -3091.226} C_VEL
LIN {X 0,Y 555.621,Z 371.276,A -85,B 0,C 180,E1 -3092.202,E2 -3092.202} C_VEL
LIN {X 0,Y 553.21,Z 371.576,A -85,B 0,C 180,E1 -3092.988,E2 -3092.988} C_VEL
LIN {X 0,Y 552.191,Z 371.704,A -85,B 0,C 180,E1 -3093.594,E2 -3093.594} C_VEL
LIN {X 0,Y 552.118,Z 371.711,A -85,B 0,C 180,E1 -3093.8,E2 -3093.8} C_VEL
LIN {X 0,Y 552.113,Z 371.714,A -85,B 0,C 180,E1 -3096.747,E2 -3096.747} C_VEL
LIN {X 0,Y 552.13,Z 371.711,A -85,B 0,C 180,E1 -3099.528,E2 -3099.528} C_VEL
LIN {X 0,Y 552.126,Z 371.713,A -85,B 0,C 180,E1 -3102.426,E2 -3102.426} C_VEL
LIN {X 0,Y 552.096,Z 371.715,A -85,B 0,C 180,E1 -3105.564,E2 -3105.564} C_VEL
LIN {X 0,Y 552.138,Z 371.71,A -85,B 0,C 180,E1 -3108.677,E2 -3108.677} C_VEL
LIN {X 0,Y 552.117,Z 371.714,A -85,B 0,C 180,E1 -3111.412,E2 -3111.412} C_VEL
LIN {X 0,Y 552.102,Z 371.715,A -85,B 0,C 180,E1 -3114.159,E2 -3114.159} C_VEL
LIN {X 0,Y 552.122,Z 371.714,A -85,B 0,C 180,E1 -3116.816,E2 -3116.816} C_VEL
LIN {X 0,Y 552.108,Z 371.715,A -85,B 0,C 180,E1 -3119.392,E2 -3119.392} C_VEL
LIN {X 0,Y 552.12,Z 371.712,A -85,B 0,C 180,E1 -3121.903,E2 -3121.903} C_VEL
LIN {X 0,Y 552.158,Z 371.709,A -85,B 0,C 180,E1 -3124.65,E2 -3124.65} C_VEL
LIN {X 0,Y 552.098,Z 371.715,A -85,B 0,C 180,E1 -3127.55,E2 -3127.55} C_VEL
LIN {X 0,Y 552.153,Z 371.707,A -85,B 0,C 180,E1 -3130.675,E2 -3130.675} C_VEL
LIN {X 0,Y 552.117,Z 371.714,A -85,B 0,C 180,E1 -3133.738,E2 -3133.738} C_VEL
LIN {X 0,Y 552.14,Z 371.71,A -85,B 0,C 180,E1 -3136.005,E2 -3136.005} C_VEL
LIN {X 0,Y 552.166,Z 371.708,A -85,B 0,C 180,E1 -3138.994,E2 -3138.994} C_VEL
LIN {X 0,Y 552.159,Z 371.708,A -85,B 0,C 180,E1 -3141.952,E2 -3141.952} C_VEL
LIN {X 0,Y 552.23,Z 371.699,A -85,B 0,C 180,E1 -3144.889,E2 -3144.889} C_VEL
LIN {X 0,Y 552.008,Z 371.73,A -85,B 0,C 180,E1 -3147.811,E2 -3147.811} C_VEL
LIN {X 0,Y 551.977,Z 371.78,A -85,B 0,C 180,E1 -3148.541,E2 -3148.541} C_VEL
LIN {X 0,Y 551.95,Z 374.273,A -85,B 0,C 180,E1 -3150.73,E2 -3150.73} C_VEL
LIN {X 0,Y 551.846,Z 378.416,A -85,B 0,C 180,E1 -3154.382,E2 -3154.382} C_VEL
LIN {X 0,Y 551.834,Z 381.697,A -85,B 0,C 180,E1 -3157.317,E2 -3157.317} C_VEL
LIN {X 0,Y 551.789,Z 385.06,A -85,B 0,C 180,E1 -3160.272,E2 -3160.272} C_VEL
LIN {X 0,Y 551.732,Z 387.581,A -85,B 0,C 180,E1 -3162.506,E2 -3162.506} C_VEL
LIN {X 0,Y 551.728,Z 390.161,A -85,B 0,C 180,E1 -3164.759,E2 -3164.759} C_VEL
LIN {X 0,Y 551.665,Z 394.02,A -85,B 0,C 180,E1 -3167.803,E2 -3167.803} C_VEL
LIN {X 0,Y 551.682,Z 395.68,A -85,B 0,C 180,E1 -3169.101,E2 -3169.101} C_VEL
LIN {X 0,Y 553.018,Z 405.082,A -85,B 0,C 180,E1 -3169.358,E2 -3169.358} C_VEL
LIN {X 0,Y 552.845,Z 417.531,A -85,B 0,C 180,E1 -3169.774,E2 -3169.774} C_VEL
LIN {X 0,Y 552.629,Z 430.478,A -85,B 0,C 180,E1 -3170.373,E2 -3170.373} C_VEL
LIN {X 0,Y 552.556,Z 441.76,A -85,B 0,C 180,E1 -3171.058,E2 -3171.058} C_VEL
LIN {X 0,Y 552.339,Z 451.982,A -85,B 0,C 180,E1 -3171.834,E2 -3171.834} C_VEL
LIN {X 0,Y 552.179,Z 460.742,A -85,B 0,C 180,E1 -3172.644,E2 -3172.644} C_VEL
LIN {X 0,Y 552.007,Z 468.893,A -85,B 0,C 180,E1 -3173.553,E2 -3173.553} C_VEL
LIN {X 0,Y 551.919,Z 476.916,A -85,B 0,C 180,E1 -3174.647,E2 -3174.647} C_VEL
LIN {X 0,Y 551.82,Z 484.025,A -85,B 0,C 180,E1 -3175.862,E2 -3175.862} C_VEL
LIN {X 0,Y 551.752,Z 488.912,A -85,B 0,C 180,E1 -3176.92,E2 -3176.92} C_VEL
LIN {X 0,Y 551.711,Z 493.165,A -85,B 0,C 180,E1 -3178.12,E2 -3178.12} C_VEL
LIN {X 0,Y 551.685,Z 495.398,A -85,B 0,C 180,E1 -3178.952,E2 -3178.952} C_VEL
LIN {X 0,Y 551.691,Z 497.38,A -85,B 0,C 180,E1 -3179.973,E2 -3179.973} C_VEL
LIN {X 0,Y 551.652,Z 498.838,A -85,B 0,C 180,E1 -3181.397,E2 -3181.397} C_VEL
LIN {X 0,Y 551.675,Z 498.786,A -85,B 0,C 180,E1 -3182.775,E2 -3182.775} C_VEL
LIN {X 0,Y 551.664,Z 497.407,A -85,B 0,C 180,E1 -3184.098,E2 -3184.098} C_VEL
LIN {X 0,Y 551.71,Z 494.791,A -85,B 0,C 180,E1 -3185.385,E2 -3185.385} C_VEL
LIN {X 0,Y 551.762,Z 490.454,A -85,B 0,C 180,E1 -3186.773,E2 -3186.773} C_VEL
LIN {X 0,Y 551.781,Z 485.928,A -85,B 0,C 180,E1 -3187.843,E2 -3187.843} C_VEL
LIN {X 0,Y 551.848,Z 479.546,A -85,B 0,C 180,E1 -3189.026,E2 -3189.026} C_VEL
LIN {X 0,Y 552.005,Z 471.641,A -85,B 0,C 180,E1 -3190.19,E2 -3190.19} C_VEL
LIN {X 0,Y 552.117,Z 463.64,A -85,B 0,C 180,E1 -3191.145,E2 -3191.145} C_VEL
LIN {X 0,Y 552.274,Z 454.466,A -85,B 0,C 180,E1 -3192.042,E2 -3192.042} C_VEL
LIN {X 0,Y 552.423,Z 444.448,A -85,B 0,C 180,E1 -3192.843,E2 -3192.843} C_VEL
LIN {X 0,Y 552.564,Z 432.41,A -85,B 0,C 180,E1 -3193.613,E2 -3193.613} C_VEL
LIN {X 0,Y 552.779,Z 420.585,A -85,B 0,C 180,E1 -3194.192,E2 -3194.192} C_VEL
LIN {X 0,Y 552.972,Z 407.41,A -85,B 0,C 180,E1 -3194.664,E2 -3194.664} C_VEL
LIN {X 0,Y 552.798,Z 402.637,A -85,B 0,C 180,E1 -3194.799,E2 -3194.799} C_VEL
LIN {X 0,Y 551.635,Z 395.666,A -85,B 0,C 180,E1 -3195.001,E2 -3195.001} C_VEL
LIN {X 0,Y 551.64,Z 392.3,A -85,B 0,C 180,E1 -3197.639,E2 -3197.639} C_VEL
LIN {X 0,Y 551.649,Z 388.913,A -85,B 0,C 180,E1 -3200.431,E2 -3200.431} C_VEL
LIN {X 0,Y 551.709,Z 385.698,A -85,B 0,C 180,E1 -3203.371,E2 -3203.371} C_VEL
LIN {X 0,Y 551.784,Z 382.843,A -85,B 0,C 180,E1 -3205.915,E2 -3205.915} C_VEL
LIN {X 0,Y 551.862,Z 379.946,A -85,B 0,C 180,E1 -3208.565,E2 -3208.565} C_VEL
LIN {X 0,Y 551.859,Z 376.663,A -85,B 0,C 180,E1 -3211.487,E2 -3211.487} C_VEL
LIN {X 0,Y 551.92,Z 373.086,A -85,B 0,C 180,E1 -3214.699,E2 -3214.699} C_VEL
LIN {X 0,Y 551.912,Z 371.741,A -85,B 0,C 180,E1 -3215.953,E2 -3215.953} C_VEL
LIN {X 0,Y 552.12,Z 371.715,A -85,B 0,C 180,E1 -3218.337,E2 -3218.337} C_VEL
LIN {X 0,Y 552.152,Z 371.709,A -85,B 0,C 180,E1 -3220.674,E2 -3220.674} C_VEL
LIN {X 0,Y 552.111,Z 371.713,A -85,B 0,C 180,E1 -3223.737,E2 -3223.737} C_VEL
LIN {X 0,Y 552.129,Z 371.712,A -85,B 0,C 180,E1 -3226.004,E2 -3226.004} C_VEL
LIN {X 0,Y 552.171,Z 371.705,A -85,B 0,C 180,E1 -3228.993,E2 -3228.993} C_VEL
LIN {X 0,Y 552.153,Z 371.709,A -85,B 0,C 180,E1 -3231.951,E2 -3231.951} C_VEL
LIN {X 0,Y 552.228,Z 371.697,A -85,B 0,C 180,E1 -3234.889,E2 -3234.889} C_VEL
LIN {X 0,Y 552.219,Z 371.701,A -85,B 0,C 180,E1 -3237.812,E2 -3237.812} C_VEL
LIN {X 0,Y 552.241,Z 371.697,A -85,B 0,C 180,E1 -3240.729,E2 -3240.729} C_VEL
LIN {X 0,Y 552.201,Z 371.703,A -85,B 0,C 180,E1 -3242.918,E2 -3242.918} C_VEL
LIN {X 0,Y 552.192,Z 371.702,A -85,B 0,C 180,E1 -3245.844,E2 -3245.844} C_VEL
LIN {X 0,Y 552.155,Z 371.71,A -85,B 0,C 180,E1 -3248.786,E2 -3248.786} C_VEL
LIN {X 0,Y 552.158,Z 371.707,A -85,B 0,C 180,E1 -3251.751,E2 -3251.751} C_VEL
LIN {X 0,Y 552.13,Z 371.712,A -85,B 0,C 180,E1 -3254.749,E2 -3254.749} C_VEL
LIN {X 0,Y 552.11,Z 371.713,A -85,B 0,C 180,E1 -3257.789,E2 -3257.789} C_VEL
LIN {X 0,Y 552.125,Z 371.711,A -85,B 0,C 180,E1 -3260.101,E2 -3260.101} C_VEL
LIN {X 0,Y 552.09,Z 371.716,A -85,B 0,C 180,E1 -3262.451,E2 -3262.451} C_VEL
LIN {X 0,Y 552.152,Z 371.708,A -85,B 0,C 180,E1 -3265.351,E2 -3265.351} C_VEL
LIN {X 0,Y 552.122,Z 371.714,A -85,B 0,C 180,E1 -3268.098,E2 -3268.098} C_VEL
LIN {X 0,Y 552.097,Z 371.718,A -85,B 0,C 180,E1 -3270.61,E2 -3270.61} C_VEL
LIN {X 0,Y 552.102,Z 371.717,A -85,B 0,C 180,E1 -3273.187,E2 -3273.187} C_VEL
LIN {X 0,Y 552.082,Z 371.718,A -85,B 0,C 180,E1 -3275.844,E2 -3275.844} C_VEL
LIN {X 0,Y 552.123,Z 371.715,A -85,B 0,C 180,E1 -3279.062,E2 -3279.062} C_VEL
LIN {X 0,Y 552.137,Z 371.713,A -85,B 0,C 180,E1 -3281.445,E2 -3281.445} C_VEL
LIN {X 0,Y 552.092,Z 371.715,A -85,B 0,C 180,E1 -3284.532,E2 -3284.532} C_VEL
LIN {X 0,Y 552.129,Z 371.714,A -85,B 0,C 180,E1 -3287.585,E2 -3287.585} C_VEL
LIN {X 0,Y 552.132,Z 371.712,A -85,B 0,C 180,E1 -3290.474,E2 -3290.474} C_VEL
LIN {X 0,Y 552.129,Z 371.758,A -85,B 0,C 180,E1 -3292.512,E2 -3292.512} C_VEL
LIN {X 0,Y 552.947,Z 376.594,A -85,B 0,C 180,E1 -3294.221,E2 -3294.221} C_VEL
LIN {X 0,Y 552.85,Z 384.509,A -85,B 0,C 180,E1 -3296.864,E2 -3296.864} C_VEL
LIN {X 0,Y 552.656,Z 393.796,A -85,B 0,C 180,E1 -3299.853,E2 -3299.853} C_VEL
LIN {X 0,Y 552.47,Z 403.044,A -85,B 0,C 180,E1 -3302.745,E2 -3302.745} C_VEL
LIN {X 0,Y 552.362,Z 410.987,A -85,B 0,C 180,E1 -3305.174,E2 -3305.174} C_VEL
LIN {X 0,Y 552.21,Z 421.578,A -85,B 0,C 180,E1 -3308.341,E2 -3308.341} C_VEL
LIN {X 0,Y 552.09,Z 430.845,A -85,B 0,C 180,E1 -3311.058,E2 -3311.058} C_VEL
LIN {X 0,Y 551.995,Z 441.436,A -85,B 0,C 180,E1 -3314.113,E2 -3314.113} C_VEL
LIN {X 0,Y 551.889,Z 451.53,A -85,B 0,C 180,E1 -3316.983,E2 -3316.983} C_VEL
LIN {X 0,Y 553.1,Z 460.526,A -85,B 0,C 180,E1 -3317.199,E2 -3317.199} C_VEL
LIN {X 0,Y 552.923,Z 473.179,A -85,B 0,C 180,E1 -3317.568,E2 -3317.568} C_VEL
LIN {X 0,Y 552.756,Z 485.486,A -85,B 0,C 180,E1 -3318.076,E2 -3318.076} C_VEL
LIN {X 0,Y 552.584,Z 497.21,A -85,B 0,C 180,E1 -3318.716,E2 -3318.716} C_VEL
LIN {X 0,Y 552.432,Z 507.928,A -85,B 0,C 180,E1 -3319.463,E2 -3319.463} C_VEL
LIN {X 0,Y 552.233,Z 517.601,A -85,B 0,C 180,E1 -3320.292,E2 -3320.292} C_VEL
LIN {X 0,Y 552.079,Z 526.413,A -85,B 0,C 180,E1 -3321.213,E2 -3321.213} C_VEL
LIN {X 0,Y 551.949,Z 535,A -85,B 0,C 180,E1 -3322.317,E2 -3322.317} C_VEL
LIN {X 0,Y 551.823,Z 541.867,A -85,B 0,C 180,E1 -3323.418,E2 -3323.418} C_VEL
LIN {X 0,Y 551.804,Z 547.365,A -85,B 0,C 180,E1 -3324.519,E2 -3324.519} C_VEL
LIN {X 0,Y 551.764,Z 551.677,A -85,B 0,C 180,E1 -3325.617,E2 -3325.617} C_VEL
LIN {X 0,Y 551.75,Z 553.957,A -85,B 0,C 180,E1 -3326.348,E2 -3326.348} C_VEL
LIN {X 0,Y 551.723,Z 555.808,A -85,B 0,C 180,E1 -3327.079,E2 -3327.079} C_VEL
LIN {X 0,Y 551.657,Z 557.199,A -85,B 0,C 180,E1 -3327.81,E2 -3327.81} C_VEL
LIN {X 0,Y 551.641,Z 558.785,A -85,B 0,C 180,E1 -3329.27,E2 -3329.27} C_VEL
LIN {X 0,Y 551.64,Z 559,A -85,B 0,C 180,E1 -3330,E2 -3330} C_VEL
LIN {X 0,Y 551.645,Z 558.186,A -85,B 0,C 180,E1 -3331.46,E2 -3331.46} C_VEL
LIN {X 0,Y 551.657,Z 557.201,A -85,B 0,C 180,E1 -3332.19,E2 -3332.19} C_VEL
LIN {X 0,Y 551.723,Z 555.81,A -85,B 0,C 180,E1 -3332.92,E2 -3332.92} C_VEL
LIN {X 0,Y 551.764,Z 552.897,A -85,B 0,C 180,E1 -3334.017,E2 -3334.017} C_VEL
LIN {X 0,Y 551.723,Z 548.95,A -85,B 0,C 180,E1 -3335.115,E2 -3335.115} C_VEL
LIN {X 0,Y 551.803,Z 543.19,A -85,B 0,C 180,E1 -3336.341,E2 -3336.341} C_VEL
LIN {X 0,Y 551.926,Z 536.239,A -85,B 0,C 180,E1 -3337.499,E2 -3337.499} C_VEL
LIN {X 0,Y 552.082,Z 527.993,A -85,B 0,C 180,E1 -3338.602,E2 -3338.602} C_VEL
LIN {X 0,Y 552.201,Z 519.542,A -85,B 0,C 180,E1 -3339.523,E2 -3339.523} C_VEL
LIN {X 0,Y 552.405,Z 509.101,A -85,B 0,C 180,E1 -3340.445,E2 -3340.445} C_VEL
LIN {X 0,Y 552.564,Z 498.297,A -85,B 0,C 180,E1 -3341.214,E2 -3341.214} C_VEL
LIN {X 0,Y 552.7,Z 487.42,A -85,B 0,C 180,E1 -3341.832,E2 -3341.832} C_VEL
LIN {X 0,Y 552.878,Z 475.775,A -85,B 0,C 180,E1 -3342.34,E2 -3342.34} C_VEL
LIN {X 0,Y 553.068,Z 462.367,A -85,B 0,C 180,E1 -3342.755,E2 -3342.755} C_VEL
LIN {X 0,Y 552.894,Z 457.823,A -85,B 0,C 180,E1 -3342.864,E2 -3342.864} C_VEL
LIN {X 0,Y 551.889,Z 451.532,A -85,B 0,C 180,E1 -3343.017,E2 -3343.017} C_VEL
LIN {X 0,Y 551.994,Z 441.437,A -85,B 0,C 180,E1 -3345.886,E2 -3345.886} C_VEL
LIN {X 0,Y 552.089,Z 430.846,A -85,B 0,C 180,E1 -3348.941,E2 -3348.941} C_VEL
LIN {X 0,Y 552.252,Z 420.257,A -85,B 0,C 180,E1 -3352.049,E2 -3352.049} C_VEL
LIN {X 0,Y 552.361,Z 410.988,A -85,B 0,C 180,E1 -3354.826,E2 -3354.826} C_VEL
LIN {X 0,Y 552.504,Z 401.721,A -85,B 0,C 180,E1 -3357.663,E2 -3357.663} C_VEL
LIN {X 0,Y 552.664,Z 392.454,A -85,B 0,C 180,E1 -3360.574,E2 -3360.574} C_VEL
LIN {X 0,Y 552.848,Z 384.511,A -85,B 0,C 180,E1 -3363.135,E2 -3363.135} C_VEL
LIN {X 0,Y 552.92,Z 376.467,A -85,B 0,C 180,E1 -3365.78,E2 -3365.78} C_VEL
LIN {X 0,Y 552.101,Z 371.717,A -85,B 0,C 180,E1 -3367.518,E2 -3367.518} C_VEL
LIN {X 0,Y 552.106,Z 371.715,A -85,B 0,C 180,E1 -3370.48,E2 -3370.48} C_VEL
LIN {X 0,Y 552.102,Z 371.715,A -85,B 0,C 180,E1 -3373.482,E2 -3373.482} C_VEL
LIN {X 0,Y 552.101,Z 371.715,A -85,B 0,C 180,E1 -3376.575,E2 -3376.575} C_VEL
LIN {X 0,Y 552.136,Z 371.713,A -85,B 0,C 180,E1 -3379.521,E2 -3379.521} C_VEL
LIN {X 0,Y 552.088,Z 371.716,A -85,B 0,C 180,E1 -3382.336,E2 -3382.336} C_VEL
LIN {X 0,Y 552.125,Z 371.714,A -85,B 0,C 180,E1 -3385.054,E2 -3385.054} C_VEL
LIN {X 0,Y 552.121,Z 371.711,A -85,B 0,C 180,E1 -3387.682,E2 -3387.682} C_VEL
LIN {X 0,Y 552.105,Z 371.713,A -85,B 0,C 180,E1 -3390.235,E2 -3390.235} C_VEL
LIN {X 0,Y 552.14,Z 371.711,A -85,B 0,C 180,E1 -3392.997,E2 -3392.997} C_VEL
LIN {X 0,Y 552.105,Z 371.715,A -85,B 0,C 180,E1 -3395.161,E2 -3395.161} C_VEL
LIN {X 0,Y 552.088,Z 371.716,A -85,B 0,C 180,E1 -3397.549,E2 -3397.549} C_VEL
LIN {X 0,Y 552.141,Z 371.71,A -85,B 0,C 180,E1 -3400.373,E2 -3400.373} C_VEL
LIN {X 0,Y 552.15,Z 371.709,A -85,B 0,C 180,E1 -3402.977,E2 -3402.977} C_VEL
LIN {X 0,Y 552.127,Z 371.712,A -85,B 0,C 180,E1 -3406.004,E2 -3406.004} C_VEL
LIN {X 0,Y 552.169,Z 371.706,A -85,B 0,C 180,E1 -3408.994,E2 -3408.994} C_VEL
LIN {X 0,Y 552.157,Z 371.708,A -85,B 0,C 180,E1 -3411.952,E2 -3411.952} C_VEL
LIN {X 0,Y 552.219,Z 371.702,A -85,B 0,C 180,E1 -3414.889,E2 -3414.889} C_VEL
LIN {X 0,Y 552.214,Z 371.699,A -85,B 0,C 180,E1 -3417.812,E2 -3417.812} C_VEL
LIN {X 0,Y 552.24,Z 371.698,A -85,B 0,C 180,E1 -3420.729,E2 -3420.729} C_VEL
LIN {X 0,Y 552.202,Z 371.703,A -85,B 0,C 180,E1 -3422.918,E2 -3422.918} C_VEL
LIN {X 0,Y 552.193,Z 371.703,A -85,B 0,C 180,E1 -3425.844,E2 -3425.844} C_VEL
LIN {X 0,Y 552.164,Z 371.707,A -85,B 0,C 180,E1 -3428.786,E2 -3428.786} C_VEL
LIN {X 0,Y 552.155,Z 371.709,A -85,B 0,C 180,E1 -3431.751,E2 -3431.751} C_VEL
LIN {X 0,Y 552.127,Z 371.713,A -85,B 0,C 180,E1 -3434.749,E2 -3434.749} C_VEL
LIN {X 0,Y 552.107,Z 371.713,A -85,B 0,C 180,E1 -3437.789,E2 -3437.789} C_VEL
LIN {X 0,Y 552.127,Z 371.712,A -85,B 0,C 180,E1 -3440.102,E2 -3440.102} C_VEL
LIN {X 0,Y 552.089,Z 371.717,A -85,B 0,C 180,E1 -3442.451,E2 -3442.451} C_VEL
LIN {X 0,Y 552.149,Z 371.707,A -85,B 0,C 180,E1 -3445.352,E2 -3445.352} C_VEL
LIN {X 0,Y 552.121,Z 371.714,A -85,B 0,C 180,E1 -3448.098,E2 -3448.098} C_VEL
LIN {X 0,Y 552.1,Z 371.715,A -85,B 0,C 180,E1 -3450.62,E2 -3450.62} C_VEL
LIN {X 0,Y 552.123,Z 371.711,A -85,B 0,C 180,E1 -3453.186,E2 -3453.186} C_VEL
LIN {X 0,Y 552.118,Z 371.711,A -85,B 0,C 180,E1 -3453.8,E2 -3453.8} C_VEL
LIN {X 0,Y 551.484,Z 371.793,A -85,B 0,C 180,E1 -3454.408,E2 -3454.408} C_VEL
LIN {X 0,Y 548.662,Z 372.148,A -85,B 0,C 180,E1 -3455.397,E2 -3455.397} C_VEL
LIN {X 0,Y 546.238,Z 372.45,A -85,B 0,C 180,E1 -3456.192,E2 -3456.192} C_VEL
LIN {X 0,Y 545.166,Z 372.581,A -85,B 0,C 180,E1 -3456.806,E2 -3456.806} C_VEL
LIN {X 0,Y 545.064,Z 372.592,A -85,B 0,C 180,E1 -3457.014,E2 -3457.014} C_VEL
LIN {X 0,Y 545.088,Z 372.589,A -85,B 0,C 180,E1 -3460.141,E2 -3460.141} C_VEL
LIN {X 0,Y 545.074,Z 372.589,A -85,B 0,C 180,E1 -3463.107,E2 -3463.107} C_VEL
LIN {X 0,Y 545.055,Z 372.593,A -85,B 0,C 180,E1 -3466.226,E2 -3466.226} C_VEL
LIN {X 0,Y 545.095,Z 372.588,A -85,B 0,C 180,E1 -3468.888,E2 -3468.888} C_VEL
LIN {X 0,Y 545.051,Z 372.593,A -85,B 0,C 180,E1 -3471.764,E2 -3471.764} C_VEL
LIN {X 0,Y 545.052,Z 372.594,A -85,B 0,C 180,E1 -3474.534,E2 -3474.534} C_VEL
LIN {X 0,Y 545.081,Z 372.589,A -85,B 0,C 180,E1 -3477.213,E2 -3477.213} C_VEL
LIN {X 0,Y 545.067,Z 372.591,A -85,B 0,C 180,E1 -3479.812,E2 -3479.812} C_VEL
LIN {X 0,Y 545.089,Z 372.59,A -85,B 0,C 180,E1 -3482.345,E2 -3482.345} C_VEL
LIN {X 0,Y 545.119,Z 372.585,A -85,B 0,C 180,E1 -3484.821,E2 -3484.821} C_VEL
LIN {X 0,Y 545.046,Z 372.593,A -85,B 0,C 180,E1 -3487.243,E2 -3487.243} C_VEL
LIN {X 0,Y 545.119,Z 372.585,A -85,B 0,C 180,E1 -3490.415,E2 -3490.415} C_VEL
LIN {X 0,Y 545.068,Z 372.593,A -85,B 0,C 180,E1 -3493.522,E2 -3493.522} C_VEL
LIN {X 0,Y 545.099,Z 372.589,A -85,B 0,C 180,E1 -3495.821,E2 -3495.821} C_VEL
LIN {X 0,Y 545.122,Z 372.585,A -85,B 0,C 180,E1 -3498.85,E2 -3498.85} C_VEL
LIN {X 0,Y 545.13,Z 372.583,A -85,B 0,C 180,E1 -3501.847,E2 -3501.847} C_VEL
LIN {X 0,Y 545.206,Z 372.574,A -85,B 0,C 180,E1 -3504.823,E2 -3504.823} C_VEL
LIN {X 0,Y 544.974,Z 372.606,A -85,B 0,C 180,E1 -3507.783,E2 -3507.783} C_VEL
LIN {X 0,Y 544.953,Z 372.61,A -85,B 0,C 180,E1 -3508.522,E2 -3508.522} C_VEL
LIN {X 0,Y 544.969,Z 374.068,A -85,B 0,C 180,E1 -3510,E2 -3510} C_VEL
LIN {X 0,Y 544.722,Z 377.448,A -85,B 0,C 180,E1 -3512.958,E2 -3512.958} C_VEL
LIN {X 0,Y 544.806,Z 379.929,A -85,B 0,C 180,E1 -3515.181,E2 -3515.181} C_VEL
LIN {X 0,Y 544.767,Z 382.438,A -85,B 0,C 180,E1 -3517.412,E2 -3517.412} C_VEL
LIN {X 0,Y 544.735,Z 385.807,A -85,B 0,C 180,E1 -3520.406,E2 -3520.406} C_VEL
LIN {X 0,Y 544.616,Z 389.199,A -85,B 0,C 180,E1 -3523.431,E2 -3523.431} C_VEL
LIN {X 0,Y 544.594,Z 391.776,A -85,B 0,C 180,E1 -3525.724,E2 -3525.724} C_VEL
LIN {X 0,Y 544.559,Z 394.562,A -85,B 0,C 180,E1 -3528.043,E2 -3528.043} C_VEL
LIN {X 0,Y 544.598,Z 395.667,A -85,B 0,C 180,E1 -3528.919,E2 -3528.919} C_VEL
LIN {X 0,Y 546.094,Z 405.516,A -85,B 0,C 180,E1 -3529.207,E2 -3529.207} C_VEL
LIN {X 0,Y 545.891,Z 418.712,A -85,B 0,C 180,E1 -3529.664,E2 -3529.664} C_VEL
LIN {X 0,Y 545.671,Z 430.297,A -85,B 0,C 180,E1 -3530.213,E2 -3530.213} C_VEL
LIN {X 0,Y 545.562,Z 442.185,A -85,B 0,C 180,E1 -3530.945,E2 -3530.945} C_VEL
LIN {X 0,Y 545.333,Z 452.064,A -85,B 0,C 180,E1 -3531.709,E2 -3531.709} C_VEL
LIN {X 0,Y 545.147,Z 461.032,A -85,B 0,C 180,E1 -3532.553,E2 -3532.553} C_VEL
LIN {X 0,Y 544.93,Z 469.877,A -85,B 0,C 180,E1 -3533.566,E2 -3533.566} C_VEL
LIN {X 0,Y 544.862,Z 477.116,A -85,B 0,C 180,E1 -3534.581,E2 -3534.581} C_VEL
LIN {X 0,Y 544.774,Z 483.576,A -85,B 0,C 180,E1 -3535.693,E2 -3535.693} C_VEL
LIN {X 0,Y 544.663,Z 488.888,A -85,B 0,C 180,E1 -3536.847,E2 -3536.847} C_VEL
LIN {X 0,Y 544.615,Z 493.254,A -85,B 0,C 180,E1 -3538.1,E2 -3538.1} C_VEL
LIN {X 0,Y 544.593,Z 496.365,A -85,B 0,C 180,E1 -3539.366,E2 -3539.366} C_VEL
LIN {X 0,Y 544.596,Z 497.787,A -85,B 0,C 180,E1 -3540.218,E2 -3540.218} C_VEL
LIN {X 0,Y 544.544,Z 498.909,A -85,B 0,C 180,E1 -3541.59,E2 -3541.59} C_VEL
LIN {X 0,Y 544.574,Z 498.659,A -85,B 0,C 180,E1 -3542.98,E2 -3542.98} C_VEL
LIN {X 0,Y 544.575,Z 497.118,A -85,B 0,C 180,E1 -3544.314,E2 -3544.314} C_VEL
LIN {X 0,Y 544.612,Z 494.339,A -85,B 0,C 180,E1 -3545.61,E2 -3545.61} C_VEL
LIN {X 0,Y 544.668,Z 490.323,A -85,B 0,C 180,E1 -3546.869,E2 -3546.869} C_VEL
LIN {X 0,Y 544.732,Z 485.078,A -85,B 0,C 180,E1 -3548.093,E2 -3548.093} C_VEL
LIN {X 0,Y 544.825,Z 478.518,A -85,B 0,C 180,E1 -3549.288,E2 -3549.288} C_VEL
LIN {X 0,Y 544.973,Z 470.39,A -85,B 0,C 180,E1 -3550.459,E2 -3550.459} C_VEL
LIN {X 0,Y 545.14,Z 461.269,A -85,B 0,C 180,E1 -3551.513,E2 -3551.513} C_VEL
LIN {X 0,Y 545.292,Z 451.362,A -85,B 0,C 180,E1 -3552.443,E2 -3552.443} C_VEL
LIN {X 0,Y 545.484,Z 441.525,A -85,B 0,C 180,E1 -3553.192,E2 -3553.192} C_VEL
LIN {X 0,Y 545.674,Z 429.878,A -85,B 0,C 180,E1 -3553.899,E2 -3553.899} C_VEL
LIN {X 0,Y 545.916,Z 417.13,A -85,B 0,C 180,E1 -3554.492,E2 -3554.492} C_VEL
LIN {X 0,Y 546.029,Z 404.5,A -85,B 0,C 180,E1 -3554.912,E2 -3554.912} C_VEL
LIN {X 0,Y 544.548,Z 395.672,A -85,B 0,C 180,E1 -3555.168,E2 -3555.168} C_VEL
LIN {X 0,Y 544.563,Z 392.401,A -85,B 0,C 180,E1 -3557.848,E2 -3557.848} C_VEL
LIN {X 0,Y 544.577,Z 389.211,A -85,B 0,C 180,E1 -3560.775,E2 -3560.775} C_VEL
LIN {X 0,Y 544.635,Z 386.103,A -85,B 0,C 180,E1 -3563.588,E2 -3563.588} C_VEL
LIN {X 0,Y 544.706,Z 383.107,A -85,B 0,C 180,E1 -3566.303,E2 -3566.303} C_VEL
LIN {X 0,Y 544.783,Z 380.213,A -85,B 0,C 180,E1 -3568.934,E2 -3568.934} C_VEL
LIN {X 0,Y 544.818,Z 377.329,A -85,B 0,C 180,E1 -3571.491,E2 -3571.491} C_VEL
LIN {X 0,Y 544.875,Z 373.65,A -85,B 0,C 180,E1 -3574.808,E2 -3574.808} C_VEL
LIN {X 0,Y 544.845,Z 372.766,A -85,B 0,C 180,E1 -3575.621,E2 -3575.621} C_VEL
LIN {X 0,Y 545.057,Z 372.594,A -85,B 0,C 180,E1 -3578.18,E2 -3578.18} C_VEL
LIN {X 0,Y 545.116,Z 372.585,A -85,B 0,C 180,E1 -3580.415,E2 -3580.415} C_VEL
LIN {X 0,Y 545.068,Z 372.592,A -85,B 0,C 180,E1 -3583.521,E2 -3583.521} C_VEL
LIN {X 0,Y 545.088,Z 372.591,A -85,B 0,C 180,E1 -3585.82,E2 -3585.82} C_VEL
LIN {X 0,Y 545.126,Z 372.582,A -85,B 0,C 180,E1 -3588.849,E2 -3588.849} C_VEL
LIN {X 0,Y 545.124,Z 372.586,A -85,B 0,C 180,E1 -3591.847,E2 -3591.847} C_VEL
LIN {X 0,Y 545.203,Z 372.572,A -85,B 0,C 180,E1 -3594.823,E2 -3594.823} C_VEL
LIN {X 0,Y 545.191,Z 372.576,A -85,B 0,C 180,E1 -3597.784,E2 -3597.784} C_VEL
LIN {X 0,Y 545.21,Z 372.572,A -85,B 0,C 180,E1 -3600.739,E2 -3600.739} C_VEL
LIN {X 0,Y 545.168,Z 372.579,A -85,B 0,C 180,E1 -3602.956,E2 -3602.956} C_VEL
LIN {X 0,Y 545.163,Z 372.578,A -85,B 0,C 180,E1 -3605.92,E2 -3605.92} C_VEL
LIN {X 0,Y 545.114,Z 372.587,A -85,B 0,C 180,E1 -3608.9,E2 -3608.9} C_VEL
LIN {X 0,Y 545.13,Z 372.582,A -85,B 0,C 180,E1 -3611.904,E2 -3611.904} C_VEL
LIN {X 0,Y 545.079,Z 372.591,A -85,B 0,C 180,E1 -3614.944,E2 -3614.944} C_VEL
LIN {X 0,Y 545.077,Z 372.589,A -85,B 0,C 180,E1 -3618.026,E2 -3618.026} C_VEL
LIN {X 0,Y 545.089,Z 372.587,A -85,B 0,C 180,E1 -3620.372,E2 -3620.372} C_VEL
LIN {X 0,Y 545.085,Z 372.589,A -85,B 0,C 180,E1 -3623.559,E2 -3623.559} C_VEL
LIN {X 0,Y 545.084,Z 372.589,A -85,B 0,C 180,E1 -3626,E2 -3626} C_VEL
LIN {X 0,Y 545.086,Z 372.587,A -85,B 0,C 180,E1 -3628.749,E2 -3628.749} C_VEL
LIN {X 0,Y 545.052,Z 372.594,A -85,B 0,C 180,E1 -3631.679,E2 -3631.679} C_VEL
LIN {X 0,Y 545.056,Z 372.593,A -85,B 0,C 180,E1 -3634.565,E2 -3634.565} C_VEL
LIN {X 0,Y 545.033,Z 372.595,A -85,B 0,C 180,E1 -3637.304,E2 -3637.304} C_VEL
LIN {X 0,Y 545.089,Z 372.59,A -85,B 0,C 180,E1 -3640.141,E2 -3640.141} C_VEL
LIN {X 0,Y 545.075,Z 372.59,A -85,B 0,C 180,E1 -3643.107,E2 -3643.107} C_VEL
LIN {X 0,Y 545.054,Z 372.595,A -85,B 0,C 180,E1 -3646.226,E2 -3646.226} C_VEL
LIN {X 0,Y 545.096,Z 372.591,A -85,B 0,C 180,E1 -3648.887,E2 -3648.887} C_VEL
LIN {X 0,Y 545.051,Z 372.595,A -85,B 0,C 180,E1 -3651.763,E2 -3651.763} C_VEL
LIN {X 0,Y 545.086,Z 372.726,A -85,B 0,C 180,E1 -3652.293,E2 -3652.293} C_VEL
LIN {X 0,Y 546.01,Z 378.018,A -85,B 0,C 180,E1 -3654.185,E2 -3654.185} C_VEL
LIN {X 0,Y 545.887,Z 385.784,A -85,B 0,C 180,E1 -3656.808,E2 -3656.808} C_VEL
LIN {X 0,Y 545.674,Z 394.477,A -85,B 0,C 180,E1 -3659.647,E2 -3659.647} C_VEL
LIN {X 0,Y 545.501,Z 403.044,A -85,B 0,C 180,E1 -3662.367,E2 -3662.367} C_VEL
LIN {X 0,Y 545.353,Z 410.987,A -85,B 0,C 180,E1 -3664.832,E2 -3664.832} C_VEL
LIN {X 0,Y 545.215,Z 421.578,A -85,B 0,C 180,E1 -3668.049,E2 -3668.049} C_VEL
LIN {X 0,Y 545.07,Z 430.845,A -85,B 0,C 180,E1 -3670.805,E2 -3670.805} C_VEL
LIN {X 0,Y 544.938,Z 441.436,A -85,B 0,C 180,E1 -3673.902,E2 -3673.902} C_VEL
LIN {X 0,Y 544.805,Z 451.53,A -85,B 0,C 180,E1 -3676.811,E2 -3676.811} C_VEL
LIN {X 0,Y 546.18,Z 461.441,A -85,B 0,C 180,E1 -3677.057,E2 -3677.057} C_VEL
LIN {X 0,Y 545.976,Z 474.476,A -85,B 0,C 180,E1 -3677.454,E2 -3677.454} C_VEL
LIN {X 0,Y 545.803,Z 485.487,A -85,B 0,C 180,E1 -3677.922,E2 -3677.922} C_VEL
LIN {X 0,Y 545.593,Z 497.594,A -85,B 0,C 180,E1 -3678.594,E2 -3678.594} C_VEL
LIN {X 0,Y 545.42,Z 509.098,A -85,B 0,C 180,E1 -3679.419,E2 -3679.419} C_VEL
LIN {X 0,Y 545.165,Z 519.538,A -85,B 0,C 180,E1 -3680.352,E2 -3680.352} C_VEL
LIN {X 0,Y 545.029,Z 527.99,A -85,B 0,C 180,E1 -3681.285,E2 -3681.285} C_VEL
LIN {X 0,Y 544.859,Z 536.237,A -85,B 0,C 180,E1 -3682.403,E2 -3682.403} C_VEL
LIN {X 0,Y 544.734,Z 543.616,A -85,B 0,C 180,E1 -3683.655,E2 -3683.655} C_VEL
LIN {X 0,Y 544.653,Z 548.95,A -85,B 0,C 180,E1 -3684.818,E2 -3684.818} C_VEL
LIN {X 0,Y 544.684,Z 552.895,A -85,B 0,C 180,E1 -3685.93,E2 -3685.93} C_VEL
LIN {X 0,Y 544.65,Z 555.808,A -85,B 0,C 180,E1 -3687.041,E2 -3687.041} C_VEL
LIN {X 0,Y 544.546,Z 558.185,A -85,B 0,C 180,E1 -3688.521,E2 -3688.521} C_VEL
LIN {X 0,Y 544.541,Z 559,A -85,B 0,C 180,E1 -3690,E2 -3690} C_VEL
LIN {X 0,Y 544.546,Z 558.186,A -85,B 0,C 180,E1 -3691.479,E2 -3691.479} C_VEL
LIN {X 0,Y 544.65,Z 555.81,A -85,B 0,C 180,E1 -3692.958,E2 -3692.958} C_VEL
LIN {X 0,Y 544.684,Z 552.897,A -85,B 0,C 180,E1 -3694.069,E2 -3694.069} C_VEL
LIN {X 0,Y 544.653,Z 548.95,A -85,B 0,C 180,E1 -3695.182,E2 -3695.182} C_VEL
LIN {X 0,Y 544.739,Z 543.704,A -85,B 0,C 180,E1 -3696.328,E2 -3696.328} C_VEL
LIN {X 0,Y 544.836,Z 537.471,A -85,B 0,C 180,E1 -3697.411,E2 -3697.411} C_VEL
LIN {X 0,Y 545.006,Z 529.481,A -85,B 0,C 180,E1 -3698.528,E2 -3698.528} C_VEL
LIN {X 0,Y 545.142,Z 521.34,A -85,B 0,C 180,E1 -3699.46,E2 -3699.46} C_VEL
LIN {X 0,Y 545.349,Z 511.406,A -85,B 0,C 180,E1 -3700.394,E2 -3700.394} C_VEL
LIN {X 0,Y 545.549,Z 501.592,A -85,B 0,C 180,E1 -3701.141,E2 -3701.141} C_VEL
LIN {X 0,Y 545.698,Z 489.186,A -85,B 0,C 180,E1 -3701.891,E2 -3701.891} C_VEL
LIN {X 0,Y 545.932,Z 476.992,A -85,B 0,C 180,E1 -3702.452,E2 -3702.452} C_VEL
LIN {X 0,Y 546.114,Z 464.194,A -85,B 0,C 180,E1 -3702.873,E2 -3702.873} C_VEL
LIN {X 0,Y 545.927,Z 458.39,A -85,B 0,C 180,E1 -3703.019,E2 -3703.019} C_VEL
LIN {X 0,Y 544.805,Z 451.532,A -85,B 0,C 180,E1 -3703.189,E2 -3703.189} C_VEL
LIN {X 0,Y 544.938,Z 441.437,A -85,B 0,C 180,E1 -3706.098,E2 -3706.098} C_VEL
LIN {X 0,Y 545.069,Z 430.846,A -85,B 0,C 180,E1 -3709.195,E2 -3709.195} C_VEL
LIN {X 0,Y 545.213,Z 421.579,A -85,B 0,C 180,E1 -3711.951,E2 -3711.951} C_VEL
LIN {X 0,Y 545.352,Z 410.988,A -85,B 0,C 180,E1 -3715.167,E2 -3715.167} C_VEL
LIN {X 0,Y 545.547,Z 401.721,A -85,B 0,C 180,E1 -3718.047,E2 -3718.047} C_VEL
LIN {X 0,Y 545.7,Z 392.454,A -85,B 0,C 180,E1 -3721.007,E2 -3721.007} C_VEL
LIN {X 0,Y 545.934,Z 384.464,A -85,B 0,C 180,E1 -3723.61,E2 -3723.61} C_VEL
LIN {X 0,Y 545.988,Z 377.85,A -85,B 0,C 180,E1 -3725.812,E2 -3725.812} C_VEL
LIN {X 0,Y 545.05,Z 372.595,A -85,B 0,C 180,E1 -3727.768,E2 -3727.768} C_VEL
LIN {X 0,Y 545.078,Z 372.59,A -85,B 0,C 180,E1 -3730.472,E2 -3730.472} C_VEL
LIN {X 0,Y 545.077,Z 372.591,A -85,B 0,C 180,E1 -3733.105,E2 -3733.105} C_VEL
LIN {X 0,Y 545.062,Z 372.594,A -85,B 0,C 180,E1 -3736.223,E2 -3736.223} C_VEL
LIN {X 0,Y 545.096,Z 372.587,A -85,B 0,C 180,E1 -3738.887,E2 -3738.887} C_VEL
LIN {X 0,Y 545.049,Z 372.596,A -85,B 0,C 180,E1 -3741.762,E2 -3741.762} C_VEL
LIN {X 0,Y 545.059,Z 372.591,A -85,B 0,C 180,E1 -3744.533,E2 -3744.533} C_VEL
LIN {X 0,Y 545.076,Z 372.592,A -85,B 0,C 180,E1 -3747.212,E2 -3747.212} C_VEL
LIN {X 0,Y 545.059,Z 372.591,A -85,B 0,C 180,E1 -3749.81,E2 -3749.81} C_VEL
LIN {X 0,Y 545.089,Z 372.588,A -85,B 0,C 180,E1 -3752.344,E2 -3752.344} C_VEL
LIN {X 0,Y 545.11,Z 372.586,A -85,B 0,C 180,E1 -3754.82,E2 -3754.82} C_VEL
LIN {X 0,Y 545.037,Z 372.596,A -85,B 0,C 180,E1 -3757.242,E2 -3757.242} C_VEL
LIN {X 0,Y 545.112,Z 372.586,A -85,B 0,C 180,E1 -3760.415,E2 -3760.415} C_VEL
LIN {X 0,Y 545.069,Z 372.59,A -85,B 0,C 180,E1 -3763.521,E2 -3763.521} C_VEL
LIN {X 0,Y 545.086,Z 372.588,A -85,B 0,C 180,E1 -3765.82,E2 -3765.82} C_VEL
LIN {X 0,Y 545.123,Z 372.584,A -85,B 0,C 180,E1 -3768.849,E2 -3768.849} C_VEL
LIN {X 0,Y 545.127,Z 372.584,A -85,B 0,C 180,E1 -3771.847,E2 -3771.847} C_VEL
LIN {X 0,Y 545.195,Z 372.577,A -85,B 0,C 180,E1 -3774.823,E2 -3774.823} C_VEL
LIN {X 0,Y 545.186,Z 372.575,A -85,B 0,C 180,E1 -3777.784,E2 -3777.784} C_VEL
LIN {X 0,Y 545.21,Z 372.574,A -85,B 0,C 180,E1 -3780.739,E2 -3780.739} C_VEL
LIN {X 0,Y 545.168,Z 372.578,A -85,B 0,C 180,E1 -3782.956,E2 -3782.956} C_VEL
LIN {X 0,Y 545.165,Z 372.579,A -85,B 0,C 180,E1 -3785.92,E2 -3785.92} C_VEL
LIN {X 0,Y 545.121,Z 372.584,A -85,B 0,C 180,E1 -3788.9,E2 -3788.9} C_VEL
LIN {X 0,Y 545.127,Z 372.584,A -85,B 0,C 180,E1 -3791.904,E2 -3791.904} C_VEL
LIN {X 0,Y 545.077,Z 372.591,A -85,B 0,C 180,E1 -3794.944,E2 -3794.944} C_VEL
LIN {X 0,Y 545.075,Z 372.59,A -85,B 0,C 180,E1 -3798.026,E2 -3798.026} C_VEL
LIN {X 0,Y 545.091,Z 372.59,A -85,B 0,C 180,E1 -3800.372,E2 -3800.372} C_VEL
LIN {X 0,Y 545.084,Z 372.589,A -85,B 0,C 180,E1 -3803.559,E2 -3803.559} C_VEL
LIN {X 0,Y 545.082,Z 372.591,A -85,B 0,C 180,E1 -3806.001,E2 -3806.001} C_VEL
LIN {X 0,Y 545.084,Z 372.589,A -85,B 0,C 180,E1 -3808.749,E2 -3808.749} C_VEL
LIN {X 0,Y 545.071,Z 372.591,A -85,B 0,C 180,E1 -3811.683,E2 -3811.683} C_VEL
LIN {X 0,Y 545.08,Z 372.59,A -85,B 0,C 180,E1 -3814.564,E2 -3814.564} C_VEL
LIN {X 0,Y 545.064,Z 372.592,A -85,B 0,C 180,E1 -3817.014,E2 -3817.014} C_VEL
LIN {X 0,Y 544.356,Z 372.679,A -85,B 0,C 180,E1 -3817.63,E2 -3817.63} C_VEL
LIN {X 0,Y 541.501,Z 373.035,A -85,B 0,C 180,E1 -3818.631,E2 -3818.631} C_VEL
LIN {X 0,Y 539.123,Z 373.332,A -85,B 0,C 180,E1 -3819.437,E2 -3819.437} C_VEL
LIN {X 0,Y 538.118,Z 373.457,A -85,B 0,C 180,E1 -3820.059,E2 -3820.059} C_VEL
LIN {X 0,Y 538.043,Z 373.463,A -85,B 0,C 180,E1 -3820.27,E2 -3820.27} C_VEL
LIN {X 0,Y 538.022,Z 373.467,A -85,B 0,C 180,E1 -3822.988,E2 -3822.988} C_VEL
LIN {X 0,Y 538.022,Z 373.471,A -85,B 0,C 180,E1 -3825.927,E2 -3825.927} C_VEL
LIN {X 0,Y 538.049,Z 373.466,A -85,B 0,C 180,E1 -3829.226,E2 -3829.226} C_VEL
LIN {X 0,Y 537.991,Z 373.473,A -85,B 0,C 180,E1 -3832.123,E2 -3832.123} C_VEL
LIN {X 0,Y 538.011,Z 373.47,A -85,B 0,C 180,E1 -3834.918,E2 -3834.918} C_VEL
LIN {X 0,Y 538.026,Z 373.468,A -85,B 0,C 180,E1 -3837.619,E2 -3837.619} C_VEL
LIN {X 0,Y 538.019,Z 373.471,A -85,B 0,C 180,E1 -3840.24,E2 -3840.24} C_VEL
LIN {X 0,Y 538.063,Z 373.462,A -85,B 0,C 180,E1 -3842.797,E2 -3842.797} C_VEL
LIN {X 0,Y 538.051,Z 373.464,A -85,B 0,C 180,E1 -3845.293,E2 -3845.293} C_VEL
LIN {X 0,Y 538.018,Z 373.471,A -85,B 0,C 180,E1 -3848.043,E2 -3848.043} C_VEL
LIN {X 0,Y 538.035,Z 373.466,A -85,B 0,C 180,E1 -3850.941,E2 -3850.941} C_VEL
LIN {X 0,Y 538.02,Z 373.468,A -85,B 0,C 180,E1 -3853.299,E2 -3853.299} C_VEL
LIN {X 0,Y 538.068,Z 373.464,A -85,B 0,C 180,E1 -3855.631,E2 -3855.631} C_VEL
LIN {X 0,Y 538.081,Z 373.461,A -85,B 0,C 180,E1 -3858.702,E2 -3858.702} C_VEL
LIN {X 0,Y 538.087,Z 373.46,A -85,B 0,C 180,E1 -3861.74,E2 -3861.74} C_VEL
LIN {X 0,Y 538.164,Z 373.451,A -85,B 0,C 180,E1 -3864.755,E2 -3864.755} C_VEL
LIN {X 0,Y 537.929,Z 373.484,A -85,B 0,C 180,E1 -3868.503,E2 -3868.503} C_VEL
LIN {X 0,Y 537.964,Z 373.903,A -85,B 0,C 180,E1 -3869.252,E2 -3869.252} C_VEL
LIN {X 0,Y 537.681,Z 377.284,A -85,B 0,C 180,E1 -3872.247,E2 -3872.247} C_VEL
LIN {X 0,Y 537.723,Z 379.789,A -85,B 0,C 180,E1 -3874.498,E2 -3874.498} C_VEL
LIN {X 0,Y 537.701,Z 383.176,A -85,B 0,C 180,E1 -3877.51,E2 -3877.51} C_VEL
LIN {X 0,Y 537.663,Z 386.557,A -85,B 0,C 180,E1 -3880.544,E2 -3880.544} C_VEL
LIN {X 0,Y 537.557,Z 389.977,A -85,B 0,C 180,E1 -3883.611,E2 -3883.611} C_VEL
LIN {X 0,Y 537.529,Z 392.563,A -85,B 0,C 180,E1 -3885.936,E2 -3885.936} C_VEL
LIN {X 0,Y 537.483,Z 395.794,A -85,B 0,C 180,E1 -3888.758,E2 -3888.758} C_VEL
LIN {X 0,Y 539.19,Z 406.412,A -85,B 0,C 180,E1 -3889.067,E2 -3889.067} C_VEL
LIN {X 0,Y 538.954,Z 419.145,A -85,B 0,C 180,E1 -3889.521,E2 -3889.521} C_VEL
LIN {X 0,Y 538.692,Z 431.635,A -85,B 0,C 180,E1 -3890.13,E2 -3890.13} C_VEL
LIN {X 0,Y 538.563,Z 442.602,A -85,B 0,C 180,E1 -3890.83,E2 -3890.83} C_VEL
LIN {X 0,Y 538.321,Z 452.41,A -85,B 0,C 180,E1 -3891.604,E2 -3891.604} C_VEL
LIN {X 0,Y 538.107,Z 461.328,A -85,B 0,C 180,E1 -3892.459,E2 -3892.459} C_VEL
LIN {X 0,Y 537.881,Z 470.121,A -85,B 0,C 180,E1 -3893.485,E2 -3893.485} C_VEL
LIN {X 0,Y 537.786,Z 477.324,A -85,B 0,C 180,E1 -3894.514,E2 -3894.514} C_VEL
LIN {X 0,Y 537.693,Z 483.494,A -85,B 0,C 180,E1 -3895.594,E2 -3895.594} C_VEL
LIN {X 0,Y 537.573,Z 489.008,A -85,B 0,C 180,E1 -3896.81,E2 -3896.81} C_VEL
LIN {X 0,Y 537.518,Z 493.343,A -85,B 0,C 180,E1 -3898.079,E2 -3898.079} C_VEL
LIN {X 0,Y 537.504,Z 495.545,A -85,B 0,C 180,E1 -3898.932,E2 -3898.932} C_VEL
LIN {X 0,Y 537.507,Z 497.973,A -85,B 0,C 180,E1 -3900.349,E2 -3900.349} C_VEL
LIN {X 0,Y 537.455,Z 498.953,A -85,B 0,C 180,E1 -3901.791,E2 -3901.791} C_VEL
LIN {X 0,Y 537.465,Z 498.428,A -85,B 0,C 180,E1 -3903.312,E2 -3903.312} C_VEL
LIN {X 0,Y 537.476,Z 496.797,A -85,B 0,C 180,E1 -3904.534,E2 -3904.534} C_VEL
LIN {X 0,Y 537.543,Z 493.813,A -85,B 0,C 180,E1 -3905.844,E2 -3905.844} C_VEL
LIN {X 0,Y 537.58,Z 489.654,A -85,B 0,C 180,E1 -3907.11,E2 -3907.11} C_VEL
LIN {X 0,Y 537.683,Z 484.236,A -85,B 0,C 180,E1 -3908.348,E2 -3908.348} C_VEL
LIN {X 0,Y 537.788,Z 477.473,A -85,B 0,C 180,E1 -3909.553,E2 -3909.553} C_VEL
LIN {X 0,Y 537.914,Z 469.134,A -85,B 0,C 180,E1 -3910.73,E2 -3910.73} C_VEL
LIN {X 0,Y 538.13,Z 460.086,A -85,B 0,C 180,E1 -3911.763,E2 -3911.763} C_VEL
LIN {X 0,Y 538.295,Z 450.664,A -85,B 0,C 180,E1 -3912.64,E2 -3912.64} C_VEL
LIN {X 0,Y 538.493,Z 439.72,A -85,B 0,C 180,E1 -3913.46,E2 -3913.46} C_VEL
LIN {X 0,Y 538.786,Z 427.958,A -85,B 0,C 180,E1 -3914.157,E2 -3914.157} C_VEL
LIN {X 0,Y 539.029,Z 415.825,A -85,B 0,C 180,E1 -3914.706,E2 -3914.706} C_VEL
LIN {X 0,Y 539.013,Z 404.772,A -85,B 0,C 180,E1 -3915.076,E2 -3915.076} C_VEL
LIN {X 0,Y 537.464,Z 395.813,A -85,B 0,C 180,E1 -3915.354,E2 -3915.354} C_VEL
LIN {X 0,Y 537.495,Z 392.662,A -85,B 0,C 180,E1 -3918.184,E2 -3918.184} C_VEL
LIN {X 0,Y 537.507,Z 389.513,A -85,B 0,C 180,E1 -3921.126,E2 -3921.126} C_VEL
LIN {X 0,Y 537.593,Z 386.135,A -85,B 0,C 180,E1 -3924.147,E2 -3924.147} C_VEL
LIN {X 0,Y 537.657,Z 383.262,A -85,B 0,C 180,E1 -3926.779,E2 -3926.779} C_VEL
LIN {X 0,Y 537.731,Z 380.148,A -85,B 0,C 180,E1 -3929.608,E2 -3929.608} C_VEL
LIN {X 0,Y 537.758,Z 376.642,A -85,B 0,C 180,E1 -3932.779,E2 -3932.779} C_VEL
LIN {X 0,Y 537.795,Z 373.878,A -85,B 0,C 180,E1 -3935.28,E2 -3935.28} C_VEL
LIN {X 0,Y 537.935,Z 373.483,A -85,B 0,C 180,E1 -3936.924,E2 -3936.924} C_VEL
LIN {X 0,Y 538.037,Z 373.467,A -85,B 0,C 180,E1 -3939.348,E2 -3939.348} C_VEL
LIN {X 0,Y 538.048,Z 373.465,A -85,B 0,C 180,E1 -3942.517,E2 -3942.517} C_VEL
LIN {X 0,Y 538.057,Z 373.465,A -85,B 0,C 180,E1 -3945.63,E2 -3945.63} C_VEL
LIN {X 0,Y 538.083,Z 373.46,A -85,B 0,C 180,E1 -3948.702,E2 -3948.702} C_VEL
LIN {X 0,Y 538.081,Z 373.463,A -85,B 0,C 180,E1 -3951.739,E2 -3951.739} C_VEL
LIN {X 0,Y 538.159,Z 373.45,A -85,B 0,C 180,E1 -3954.755,E2 -3954.755} C_VEL
LIN {X 0,Y 538.163,Z 373.451,A -85,B 0,C 180,E1 -3957.755,E2 -3957.755} C_VEL
LIN {X 0,Y 538.18,Z 373.448,A -85,B 0,C 180,E1 -3960.748,E2 -3960.748} C_VEL
LIN {X 0,Y 538.134,Z 373.455,A -85,B 0,C 180,E1 -3962.994,E2 -3962.994} C_VEL
LIN {X 0,Y 538.116,Z 373.456,A -85,B 0,C 180,E1 -3965.997,E2 -3965.997} C_VEL
LIN {X 0,Y 538.065,Z 373.464,A -85,B 0,C 180,E1 -3969.018,E2 -3969.018} C_VEL
LIN {X 0,Y 538.078,Z 373.461,A -85,B 0,C 180,E1 -3972.063,E2 -3972.063} C_VEL
LIN {X 0,Y 538.039,Z 373.466,A -85,B 0,C 180,E1 -3975.144,E2 -3975.144} C_VEL
LIN {X 0,Y 538.029,Z 373.468,A -85,B 0,C 180,E1 -3978.27,E2 -3978.27} C_VEL
LIN {X 0,Y 538.033,Z 373.467,A -85,B 0,C 180,E1 -3980.652,E2 -3980.652} C_VEL
LIN {X 0,Y 538.019,Z 373.468,A -85,B 0,C 180,E1 -3983.888,E2 -3983.888} C_VEL
LIN {X 0,Y 538.045,Z 373.464,A -85,B 0,C 180,E1 -3986.367,E2 -3986.367} C_VEL
LIN {X 0,Y 538.026,Z 373.466,A -85,B 0,C 180,E1 -3988.934,E2 -3988.934} C_VEL
LIN {X 0,Y 538.005,Z 373.474,A -85,B 0,C 180,E1 -3991.888,E2 -3991.888} C_VEL
LIN {X 0,Y 538.006,Z 373.471,A -85,B 0,C 180,E1 -3994.618,E2 -3994.618} C_VEL
LIN {X 0,Y 538,Z 373.471,A -85,B 0,C 180,E1 -3997.17,E2 -3997.17} C_VEL
LIN {X 0,Y 538.051,Z 373.465,A -85,B 0,C 180,E1 -3999.795,E2 -3999.795} C_VEL
LIN {X 0,Y 538.016,Z 373.471,A -85,B 0,C 180,E1 -4002.786,E2 -4002.786} C_VEL
LIN {X 0,Y 538.022,Z 373.469,A -85,B 0,C 180,E1 -4005.927,E2 -4005.927} C_VEL
LIN {X 0,Y 538.051,Z 373.466,A -85,B 0,C 180,E1 -4009.253,E2 -4009.253} C_VEL
LIN {X 0,Y 538.031,Z 373.509,A -85,B 0,C 180,E1 -4011.998,E2 -4011.998} C_VEL
LIN {X 0,Y 538.993,Z 379.033,A -85,B 0,C 180,E1 -4014.073,E2 -4014.073} C_VEL
LIN {X 0,Y 538.959,Z 386.519,A -85,B 0,C 180,E1 -4016.57,E2 -4016.57} C_VEL
LIN {X 0,Y 538.72,Z 395.143,A -85,B 0,C 180,E1 -4019.432,E2 -4019.432} C_VEL
LIN {X 0,Y 538.552,Z 403.044,A -85,B 0,C 180,E1 -4021.98,E2 -4021.98} C_VEL
LIN {X 0,Y 538.329,Z 412.311,A -85,B 0,C 180,E1 -4024.894,E2 -4024.894} C_VEL
LIN {X 0,Y 538.177,Z 422.409,A -85,B 0,C 180,E1 -4028,E2 -4028} C_VEL
LIN {X 0,Y 538.025,Z 430.845,A -85,B 0,C 180,E1 -4030.543,E2 -4030.543} C_VEL
LIN {X 0,Y 537.895,Z 440.112,A -85,B 0,C 180,E1 -4033.295,E2 -4033.295} C_VEL
LIN {X 0,Y 537.785,Z 449.379,A -85,B 0,C 180,E1 -4036.009,E2 -4036.009} C_VEL
LIN {X 0,Y 537.738,Z 451.53,A -85,B 0,C 180,E1 -4036.634,E2 -4036.634} C_VEL
LIN {X 0,Y 539.252,Z 462.356,A -85,B 0,C 180,E1 -4036.912,E2 -4036.912} C_VEL
LIN {X 0,Y 539.022,Z 475.771,A -85,B 0,C 180,E1 -4037.338,E2 -4037.338} C_VEL
LIN {X 0,Y 538.817,Z 487.413,A -85,B 0,C 180,E1 -4037.859,E2 -4037.859} C_VEL
LIN {X 0,Y 538.619,Z 497.974,A -85,B 0,C 180,E1 -4038.47,E2 -4038.47} C_VEL
LIN {X 0,Y 538.387,Z 509.099,A -85,B 0,C 180,E1 -4039.28,E2 -4039.28} C_VEL
LIN {X 0,Y 538.139,Z 519.538,A -85,B 0,C 180,E1 -4040.225,E2 -4040.225} C_VEL
LIN {X 0,Y 537.974,Z 527.99,A -85,B 0,C 180,E1 -4041.17,E2 -4041.17} C_VEL
LIN {X 0,Y 537.817,Z 536.237,A -85,B 0,C 180,E1 -4042.302,E2 -4042.302} C_VEL
LIN {X 0,Y 537.683,Z 542.751,A -85,B 0,C 180,E1 -4043.409,E2 -4043.409} C_VEL
LIN {X 0,Y 537.676,Z 547.365,A -85,B 0,C 180,E1 -4044.374,E2 -4044.374} C_VEL
LIN {X 0,Y 537.558,Z 551.677,A -85,B 0,C 180,E1 -4045.501,E2 -4045.501} C_VEL
LIN {X 0,Y 537.591,Z 553.957,A -85,B 0,C 180,E1 -4046.252,E2 -4046.252} C_VEL
LIN {X 0,Y 537.551,Z 555.808,A -85,B 0,C 180,E1 -4047.002,E2 -4047.002} C_VEL
LIN {X 0,Y 537.49,Z 557.198,A -85,B 0,C 180,E1 -4047.752,E2 -4047.752} C_VEL
LIN {X 0,Y 537.442,Z 558.785,A -85,B 0,C 180,E1 -4049.251,E2 -4049.251} C_VEL
LIN {X 0,Y 537.442,Z 559,A -85,B 0,C 180,E1 -4050,E2 -4050} C_VEL
LIN {X 0,Y 537.451,Z 558.187,A -85,B 0,C 180,E1 -4051.498,E2 -4051.498} C_VEL
LIN {X 0,Y 537.49,Z 557.2,A -85,B 0,C 180,E1 -4052.248,E2 -4052.248} C_VEL
LIN {X 0,Y 537.551,Z 555.81,A -85,B 0,C 180,E1 -4052.997,E2 -4052.997} C_VEL
LIN {X 0,Y 537.603,Z 552.897,A -85,B 0,C 180,E1 -4054.123,E2 -4054.123} C_VEL
LIN {X 0,Y 537.587,Z 548.95,A -85,B 0,C 180,E1 -4055.25,E2 -4055.25} C_VEL
LIN {X 0,Y 537.65,Z 544.08,A -85,B 0,C 180,E1 -4056.335,E2 -4056.335} C_VEL
LIN {X 0,Y 537.79,Z 537.471,A -85,B 0,C 180,E1 -4057.509,E2 -4057.509} C_VEL
LIN {X 0,Y 537.972,Z 529.481,A -85,B 0,C 180,E1 -4058.64,E2 -4058.64} C_VEL
LIN {X 0,Y 538.119,Z 521.339,A -85,B 0,C 180,E1 -4059.585,E2 -4059.585} C_VEL
LIN {X 0,Y 538.342,Z 511.406,A -85,B 0,C 180,E1 -4060.531,E2 -4060.531} C_VEL
LIN {X 0,Y 538.563,Z 501.593,A -85,B 0,C 180,E1 -4061.288,E2 -4061.288} C_VEL
LIN {X 0,Y 538.717,Z 490.563,A -85,B 0,C 180,E1 -4061.973,E2 -4061.973} C_VEL
LIN {X 0,Y 538.979,Z 478.121,A -85,B 0,C 180,E1 -4062.567,E2 -4062.567} C_VEL
LIN {X 0,Y 539.185,Z 465.107,A -85,B 0,C 180,E1 -4063.017,E2 -4063.017} C_VEL
LIN {X 0,Y 539.005,Z 459.101,A -85,B 0,C 180,E1 -4063.174,E2 -4063.174} C_VEL
LIN {X 0,Y 537.738,Z 451.532,A -85,B 0,C 180,E1 -4063.365,E2 -4063.365} C_VEL
LIN {X 0,Y 537.878,Z 441.437,A -85,B 0,C 180,E1 -4066.315,E2 -4066.315} C_VEL
LIN {X 0,Y 537.999,Z 432.17,A -85,B 0,C 180,E1 -4069.061,E2 -4069.061} C_VEL
LIN {X 0,Y 538.124,Z 424.227,A -85,B 0,C 180,E1 -4071.449,E2 -4071.449} C_VEL
LIN {X 0,Y 538.313,Z 414.961,A -85,B 0,C 180,E1 -4074.282,E2 -4074.282} C_VEL
LIN {X 0,Y 538.457,Z 405.693,A -85,B 0,C 180,E1 -4077.182,E2 -4077.182} C_VEL
LIN {X 0,Y 538.63,Z 397.75,A -85,B 0,C 180,E1 -4079.723,E2 -4079.723} C_VEL
LIN {X 0,Y 538.874,Z 388.422,A -85,B 0,C 180,E1 -4082.767,E2 -4082.767} C_VEL
LIN {X 0,Y 539.037,Z 380.354,A -85,B 0,C 180,E1 -4085.463,E2 -4085.463} C_VEL
LIN {X 0,Y 538.569,Z 376.342,A -85,B 0,C 180,E1 -4086.888,E2 -4086.888} C_VEL
LIN {X 0,Y 538.019,Z 373.471,A -85,B 0,C 180,E1 -4088.067,E2 -4088.067} C_VEL
LIN {X 0,Y 538.045,Z 373.468,A -85,B 0,C 180,E1 -4090.775,E2 -4090.775} C_VEL
LIN {X 0,Y 538.022,Z 373.471,A -85,B 0,C 180,E1 -4094.073,E2 -4094.073} C_VEL
LIN {X 0,Y 538.021,Z 373.469,A -85,B 0,C 180,E1 -4097.012,E2 -4097.012} C_VEL
LIN {X 0,Y 538.073,Z 373.463,A -85,B 0,C 180,E1 -4099.248,E2 -4099.248} C_VEL
LIN {X 0,Y 537.989,Z 373.472,A -85,B 0,C 180,E1 -4102.122,E2 -4102.122} C_VEL
LIN {X 0,Y 538.015,Z 373.471,A -85,B 0,C 180,E1 -4104.917,E2 -4104.917} C_VEL
LIN {X 0,Y 538.025,Z 373.467,A -85,B 0,C 180,E1 -4107.618,E2 -4107.618} C_VEL
LIN {X 0,Y 538.011,Z 373.469,A -85,B 0,C 180,E1 -4110.238,E2 -4110.238} C_VEL
LIN {X 0,Y 538.064,Z 373.465,A -85,B 0,C 180,E1 -4112.796,E2 -4112.796} C_VEL
LIN {X 0,Y 538.041,Z 373.466,A -85,B 0,C 180,E1 -4115.292,E2 -4115.292} C_VEL
LIN {X 0,Y 538.006,Z 373.469,A -85,B 0,C 180,E1 -4118.041,E2 -4118.041} C_VEL
LIN {X 0,Y 538.033,Z 373.467,A -85,B 0,C 180,E1 -4120.94,E2 -4120.94} C_VEL
LIN {X 0,Y 538.019,Z 373.468,A -85,B 0,C 180,E1 -4123.299,E2 -4123.299} C_VEL
LIN {X 0,Y 538.054,Z 373.463,A -85,B 0,C 180,E1 -4125.63,E2 -4125.63} C_VEL
LIN {X 0,Y 538.08,Z 373.461,A -85,B 0,C 180,E1 -4128.702,E2 -4128.702} C_VEL
LIN {X 0,Y 538.083,Z 373.462,A -85,B 0,C 180,E1 -4131.74,E2 -4131.74} C_VEL
LIN {X 0,Y 538.152,Z 373.453,A -85,B 0,C 180,E1 -4134.755,E2 -4134.755} C_VEL
LIN {X 0,Y 538.158,Z 373.45,A -85,B 0,C 180,E1 -4137.755,E2 -4137.755} C_VEL
LIN {X 0,Y 538.179,Z 373.449,A -85,B 0,C 180,E1 -4140.748,E2 -4140.748} C_VEL
LIN {X 0,Y 538.134,Z 373.454,A -85,B 0,C 180,E1 -4142.995,E2 -4142.995} C_VEL
LIN {X 0,Y 538.117,Z 373.458,A -85,B 0,C 180,E1 -4145.997,E2 -4145.997} C_VEL
LIN {X 0,Y 538.07,Z 373.463,A -85,B 0,C 180,E1 -4149.018,E2 -4149.018} C_VEL
LIN {X 0,Y 538.075,Z 373.462,A -85,B 0,C 180,E1 -4152.063,E2 -4152.063} C_VEL
LIN {X 0,Y 538.037,Z 373.466,A -85,B 0,C 180,E1 -4155.144,E2 -4155.144} C_VEL
LIN {X 0,Y 538.027,Z 373.47,A -85,B 0,C 180,E1 -4158.271,E2 -4158.271} C_VEL
LIN {X 0,Y 538.035,Z 373.467,A -85,B 0,C 180,E1 -4160.652,E2 -4160.652} C_VEL
LIN {X 0,Y 538.016,Z 373.471,A -85,B 0,C 180,E1 -4163.888,E2 -4163.888} C_VEL
LIN {X 0,Y 538.043,Z 373.466,A -85,B 0,C 180,E1 -4166.367,E2 -4166.367} C_VEL
LIN {X 0,Y 538.025,Z 373.468,A -85,B 0,C 180,E1 -4168.935,E2 -4168.935} C_VEL
LIN {X 0,Y 538.021,Z 373.469,A -85,B 0,C 180,E1 -4171.891,E2 -4171.891} C_VEL
LIN {X 0,Y 538.029,Z 373.469,A -85,B 0,C 180,E1 -4174.622,E2 -4174.622} C_VEL
LIN {X 0,Y 538.006,Z 373.471,A -85,B 0,C 180,E1 -4177.172,E2 -4177.172} C_VEL
LIN {X 0,Y 538.043,Z 373.463,A -85,B 0,C 180,E1 -4180.27,E2 -4180.27} C_VEL
LIN {X 0,Y 537.39,Z 373.547,A -85,B 0,C 180,E1 -4180.895,E2 -4180.895} C_VEL
LIN {X 0,Y 534.523,Z 373.906,A -85,B 0,C 180,E1 -4181.909,E2 -4181.909} C_VEL
LIN {X 0,Y 532.086,Z 374.21,A -85,B 0,C 180,E1 -4182.726,E2 -4182.726} C_VEL
LIN {X 0,Y 531.036,Z 374.339,A -85,B 0,C 180,E1 -4183.357,E2 -4183.357} C_VEL
LIN {X 0,Y 530.948,Z 374.349,A -85,B 0,C 180,E1 -4183.571,E2 -4183.571} C_VEL
LIN {X 0,Y 530.958,Z 374.348,A -85,B 0,C 180,E1 -4186.506,E2 -4186.506} C_VEL
LIN {X 0,Y 530.987,Z 374.346,A -85,B 0,C 180,E1 -4188.977,E2 -4188.977} C_VEL
LIN {X 0,Y 530.957,Z 374.35,A -85,B 0,C 180,E1 -4191.53,E2 -4191.53} C_VEL
LIN {X 0,Y 530.975,Z 374.347,A -85,B 0,C 180,E1 -4194.383,E2 -4194.383} C_VEL
LIN {X 0,Y 530.97,Z 374.348,A -85,B 0,C 180,E1 -4197.135,E2 -4197.135} C_VEL
LIN {X 0,Y 530.97,Z 374.347,A -85,B 0,C 180,E1 -4199.804,E2 -4199.804} C_VEL
LIN {X 0,Y 531.016,Z 374.342,A -85,B 0,C 180,E1 -4202.468,E2 -4202.468} C_VEL
LIN {X 0,Y 531.008,Z 374.342,A -85,B 0,C 180,E1 -4204.943,E2 -4204.943} C_VEL
LIN {X 0,Y 530.974,Z 374.347,A -85,B 0,C 180,E1 -4208.247,E2 -4208.247} C_VEL
LIN {X 0,Y 530.995,Z 374.343,A -85,B 0,C 180,E1 -4210.678,E2 -4210.678} C_VEL
LIN {X 0,Y 530.984,Z 374.344,A -85,B 0,C 180,E1 -4213.071,E2 -4213.071} C_VEL
LIN {X 0,Y 531.023,Z 374.34,A -85,B 0,C 180,E1 -4215.436,E2 -4215.436} C_VEL
LIN {X 0,Y 531.041,Z 374.337,A -85,B 0,C 180,E1 -4218.55,E2 -4218.55} C_VEL
LIN {X 0,Y 531.056,Z 374.337,A -85,B 0,C 180,E1 -4221.63,E2 -4221.63} C_VEL
LIN {X 0,Y 531.124,Z 374.328,A -85,B 0,C 180,E1 -4224.686,E2 -4224.686} C_VEL
LIN {X 0,Y 530.904,Z 374.359,A -85,B 0,C 180,E1 -4228.483,E2 -4228.483} C_VEL
LIN {X 0,Y 530.903,Z 374.569,A -85,B 0,C 180,E1 -4229.242,E2 -4229.242} C_VEL
LIN {X 0,Y 530.69,Z 377.117,A -85,B 0,C 180,E1 -4231.518,E2 -4231.518} C_VEL
LIN {X 0,Y 530.663,Z 380.496,A -85,B 0,C 180,E1 -4234.558,E2 -4234.558} C_VEL
LIN {X 0,Y 530.671,Z 383.088,A -85,B 0,C 180,E1 -4236.846,E2 -4236.846} C_VEL
LIN {X 0,Y 530.544,Z 386.503,A -85,B 0,C 180,E1 -4239.916,E2 -4239.916} C_VEL
LIN {X 0,Y 530.518,Z 389.064,A -85,B 0,C 180,E1 -4242.237,E2 -4242.237} C_VEL
LIN {X 0,Y 530.476,Z 392.477,A -85,B 0,C 180,E1 -4245.365,E2 -4245.365} C_VEL
LIN {X 0,Y 530.41,Z 395.181,A -85,B 0,C 180,E1 -4247.743,E2 -4247.743} C_VEL
LIN {X 0,Y 530.407,Z 396.136,A -85,B 0,C 180,E1 -4248.567,E2 -4248.567} C_VEL
LIN {X 0,Y 532.28,Z 407.656,A -85,B 0,C 180,E1 -4248.924,E2 -4248.924} C_VEL
LIN {X 0,Y 532.033,Z 420.136,A -85,B 0,C 180,E1 -4249.384,E2 -4249.384} C_VEL
LIN {X 0,Y 531.751,Z 432.374,A -85,B 0,C 180,E1 -4249.997,E2 -4249.997} C_VEL
LIN {X 0,Y 531.602,Z 443.226,A -85,B 0,C 180,E1 -4250.71,E2 -4250.71} C_VEL
LIN {X 0,Y 531.298,Z 453.379,A -85,B 0,C 180,E1 -4251.535,E2 -4251.535} C_VEL
LIN {X 0,Y 531.061,Z 462.319,A -85,B 0,C 180,E1 -4252.425,E2 -4252.425} C_VEL
LIN {X 0,Y 530.827,Z 471.502,A -85,B 0,C 180,E1 -4253.547,E2 -4253.547} C_VEL
LIN {X 0,Y 530.683,Z 480.011,A -85,B 0,C 180,E1 -4254.864,E2 -4254.864} C_VEL
LIN {X 0,Y 530.575,Z 485.478,A -85,B 0,C 180,E1 -4255.92,E2 -4255.92} C_VEL
LIN {X 0,Y 530.499,Z 490.342,A -85,B 0,C 180,E1 -4257.097,E2 -4257.097} C_VEL
LIN {X 0,Y 530.422,Z 494.601,A -85,B 0,C 180,E1 -4258.489,E2 -4258.489} C_VEL
LIN {X 0,Y 530.401,Z 496.485,A -85,B 0,C 180,E1 -4259.357,E2 -4259.357} C_VEL
LIN {X 0,Y 530.383,Z 498.194,A -85,B 0,C 180,E1 -4260.536,E2 -4260.536} C_VEL
LIN {X 0,Y 530.376,Z 498.998,A -85,B 0,C 180,E1 -4262.008,E2 -4262.008} C_VEL
LIN {X 0,Y 530.361,Z 498.354,A -85,B 0,C 180,E1 -4263.401,E2 -4263.401} C_VEL
LIN {X 0,Y 530.377,Z 496.433,A -85,B 0,C 180,E1 -4264.758,E2 -4264.758} C_VEL
LIN {X 0,Y 530.482,Z 493.284,A -85,B 0,C 180,E1 -4266.084,E2 -4266.084} C_VEL
LIN {X 0,Y 530.505,Z 488.983,A -85,B 0,C 180,E1 -4267.357,E2 -4267.357} C_VEL
LIN {X 0,Y 530.58,Z 483.401,A -85,B 0,C 180,E1 -4268.601,E2 -4268.601} C_VEL
LIN {X 0,Y 530.753,Z 476.374,A -85,B 0,C 180,E1 -4269.824,E2 -4269.824} C_VEL
LIN {X 0,Y 530.905,Z 467.922,A -85,B 0,C 180,E1 -4271.013,E2 -4271.013} C_VEL
LIN {X 0,Y 531.144,Z 459.901,A -85,B 0,C 180,E1 -4271.928,E2 -4271.928} C_VEL
LIN {X 0,Y 531.309,Z 450.535,A -85,B 0,C 180,E1 -4272.809,E2 -4272.809} C_VEL
LIN {X 0,Y 531.611,Z 438.844,A -85,B 0,C 180,E1 -4273.689,E2 -4273.689} C_VEL
LIN {X 0,Y 531.873,Z 428.247,A -85,B 0,C 180,E1 -4274.32,E2 -4274.32} C_VEL
LIN {X 0,Y 532.088,Z 417.319,A -85,B 0,C 180,E1 -4274.829,E2 -4274.829} C_VEL
LIN {X 0,Y 532.091,Z 405.566,A -85,B 0,C 180,E1 -4275.237,E2 -4275.237} C_VEL
LIN {X 0,Y 530.379,Z 396.22,A -85,B 0,C 180,E1 -4275.522,E2 -4275.522} C_VEL
LIN {X 0,Y 530.416,Z 392.947,A -85,B 0,C 180,E1 -4278.509,E2 -4278.509} C_VEL
LIN {X 0,Y 530.464,Z 389.735,A -85,B 0,C 180,E1 -4281.487,E2 -4281.487} C_VEL
LIN {X 0,Y 530.521,Z 386.609,A -85,B 0,C 180,E1 -4284.346,E2 -4284.346} C_VEL
LIN {X 0,Y 530.583,Z 383.582,A -85,B 0,C 180,E1 -4287.106,E2 -4287.106} C_VEL
LIN {X 0,Y 530.667,Z 380.66,A -85,B 0,C 180,E1 -4289.784,E2 -4289.784} C_VEL
LIN {X 0,Y 530.657,Z 377.623,A -85,B 0,C 180,E1 -4292.54,E2 -4292.54} C_VEL
LIN {X 0,Y 530.717,Z 374.998,A -85,B 0,C 180,E1 -4294.928,E2 -4294.928} C_VEL
LIN {X 0,Y 530.789,Z 374.372,A -85,B 0,C 180,E1 -4296.006,E2 -4296.006} C_VEL
LIN {X 0,Y 530.964,Z 374.35,A -85,B 0,C 180,E1 -4298.246,E2 -4298.246} C_VEL
LIN {X 0,Y 530.992,Z 374.345,A -85,B 0,C 180,E1 -4300.677,E2 -4300.677} C_VEL
LIN {X 0,Y 530.98,Z 374.345,A -85,B 0,C 180,E1 -4303.071,E2 -4303.071} C_VEL
LIN {X 0,Y 531.013,Z 374.341,A -85,B 0,C 180,E1 -4305.436,E2 -4305.436} C_VEL
LIN {X 0,Y 531.04,Z 374.338,A -85,B 0,C 180,E1 -4308.55,E2 -4308.55} C_VEL
LIN {X 0,Y 531.051,Z 374.337,A -85,B 0,C 180,E1 -4311.629,E2 -4311.629} C_VEL
LIN {X 0,Y 531.118,Z 374.327,A -85,B 0,C 180,E1 -4314.685,E2 -4314.685} C_VEL
LIN {X 0,Y 531.134,Z 374.326,A -85,B 0,C 180,E1 -4317.725,E2 -4317.725} C_VEL
LIN {X 0,Y 531.15,Z 374.324,A -85,B 0,C 180,E1 -4320.758,E2 -4320.758} C_VEL
LIN {X 0,Y 531.101,Z 374.331,A -85,B 0,C 180,E1 -4323.034,E2 -4323.034} C_VEL
LIN {X 0,Y 531.076,Z 374.333,A -85,B 0,C 180,E1 -4326.077,E2 -4326.077} C_VEL
LIN {X 0,Y 531.025,Z 374.34,A -85,B 0,C 180,E1 -4329.138,E2 -4329.138} C_VEL
LIN {X 0,Y 531.035,Z 374.339,A -85,B 0,C 180,E1 -4332.225,E2 -4332.225} C_VEL
LIN {X 0,Y 530.99,Z 374.343,A -85,B 0,C 180,E1 -4335.35,E2 -4335.35} C_VEL
LIN {X 0,Y 531.011,Z 374.341,A -85,B 0,C 180,E1 -4337.723,E2 -4337.723} C_VEL
LIN {X 0,Y 530.994,Z 374.346,A -85,B 0,C 180,E1 -4340.938,E2 -4340.938} C_VEL
LIN {X 0,Y 530.975,Z 374.346,A -85,B 0,C 180,E1 -4344.225,E2 -4344.225} C_VEL
LIN {X 0,Y 531.007,Z 374.342,A -85,B 0,C 180,E1 -4346.744,E2 -4346.744} C_VEL
LIN {X 0,Y 530.977,Z 374.347,A -85,B 0,C 180,E1 -4349.323,E2 -4349.323} C_VEL
LIN {X 0,Y 530.96,Z 374.349,A -85,B 0,C 180,E1 -4352.101,E2 -4352.101} C_VEL
LIN {X 0,Y 530.965,Z 374.347,A -85,B 0,C 180,E1 -4354.852,E2 -4354.852} C_VEL
LIN {X 0,Y 530.962,Z 374.349,A -85,B 0,C 180,E1 -4357.508,E2 -4357.508} C_VEL
LIN {X 0,Y 531.023,Z 374.342,A -85,B 0,C 180,E1 -4360.429,E2 -4360.429} C_VEL
LIN {X 0,Y 530.952,Z 374.349,A -85,B 0,C 180,E1 -4363.496,E2 -4363.496} C_VEL
LIN {X 0,Y 530.957,Z 374.351,A -85,B 0,C 180,E1 -4366.505,E2 -4366.505} C_VEL
LIN {X 0,Y 530.988,Z 374.347,A -85,B 0,C 180,E1 -4368.976,E2 -4368.976} C_VEL
LIN {X 0,Y 531.001,Z 374.493,A -85,B 0,C 180,E1 -4371.776,E2 -4371.776} C_VEL
LIN {X 0,Y 532.021,Z 380.465,A -85,B 0,C 180,E1 -4374.085,E2 -4374.085} C_VEL
LIN {X 0,Y 531.984,Z 387.143,A -85,B 0,C 180,E1 -4376.335,E2 -4376.335} C_VEL
LIN {X 0,Y 531.749,Z 395.113,A -85,B 0,C 180,E1 -4378.973,E2 -4378.973} C_VEL
LIN {X 0,Y 531.558,Z 404.369,A -85,B 0,C 180,E1 -4382.008,E2 -4382.008} C_VEL
LIN {X 0,Y 531.322,Z 413.635,A -85,B 0,C 180,E1 -4384.959,E2 -4384.959} C_VEL
LIN {X 0,Y 531.161,Z 422.913,A -85,B 0,C 180,E1 -4387.85,E2 -4387.85} C_VEL
LIN {X 0,Y 530.967,Z 432.169,A -85,B 0,C 180,E1 -4390.676,E2 -4390.676} C_VEL
LIN {X 0,Y 530.826,Z 441.436,A -85,B 0,C 180,E1 -4393.462,E2 -4393.462} C_VEL
LIN {X 0,Y 530.708,Z 451.365,A -85,B 0,C 180,E1 -4396.405,E2 -4396.405} C_VEL
LIN {X 0,Y 530.697,Z 451.53,A -85,B 0,C 180,E1 -4396.454,E2 -4396.454} C_VEL
LIN {X 0,Y 532.35,Z 462.356,A -85,B 0,C 180,E1 -4396.739,E2 -4396.739} C_VEL
LIN {X 0,Y 532.107,Z 475.772,A -85,B 0,C 180,E1 -4397.17,E2 -4397.17} C_VEL
LIN {X 0,Y 531.865,Z 487.412,A -85,B 0,C 180,E1 -4397.698,E2 -4397.698} C_VEL
LIN {X 0,Y 531.642,Z 498.405,A -85,B 0,C 180,E1 -4398.346,E2 -4398.346} C_VEL
LIN {X 0,Y 531.389,Z 510.261,A -85,B 0,C 180,E1 -4399.233,E2 -4399.233} C_VEL
LIN {X 0,Y 531.114,Z 519.539,A -85,B 0,C 180,E1 -4400.095,E2 -4400.095} C_VEL
LIN {X 0,Y 530.931,Z 527.991,A -85,B 0,C 180,E1 -4401.052,E2 -4401.052} C_VEL
LIN {X 0,Y 530.758,Z 536.237,A -85,B 0,C 180,E1 -4402.199,E2 -4402.199} C_VEL
LIN {X 0,Y 530.598,Z 543.27,A -85,B 0,C 180,E1 -4403.419,E2 -4403.419} C_VEL
LIN {X 0,Y 530.524,Z 548.949,A -85,B 0,C 180,E1 -4404.679,E2 -4404.679} C_VEL
LIN {X 0,Y 530.522,Z 552.895,A -85,B 0,C 180,E1 -4405.822,E2 -4405.822} C_VEL
LIN {X 0,Y 530.457,Z 555.808,A -85,B 0,C 180,E1 -4406.962,E2 -4406.962} C_VEL
LIN {X 0,Y 530.411,Z 557.197,A -85,B 0,C 180,E1 -4407.722,E2 -4407.722} C_VEL
LIN {X 0,Y 530.344,Z 558.785,A -85,B 0,C 180,E1 -4409.241,E2 -4409.241} C_VEL
LIN {X 0,Y 530.342,Z 559,A -85,B 0,C 180,E1 -4410,E2 -4410} C_VEL
LIN {X 0,Y 530.361,Z 558.186,A -85,B 0,C 180,E1 -4411.518,E2 -4411.518} C_VEL
LIN {X 0,Y 530.411,Z 557.199,A -85,B 0,C 180,E1 -4412.278,E2 -4412.278} C_VEL
LIN {X 0,Y 530.457,Z 555.81,A -85,B 0,C 180,E1 -4413.038,E2 -4413.038} C_VEL
LIN {X 0,Y 530.522,Z 552.896,A -85,B 0,C 180,E1 -4414.178,E2 -4414.178} C_VEL
LIN {X 0,Y 530.524,Z 548.95,A -85,B 0,C 180,E1 -4415.32,E2 -4415.32} C_VEL
LIN {X 0,Y 530.599,Z 543.265,A -85,B 0,C 180,E1 -4416.582,E2 -4416.582} C_VEL
LIN {X 0,Y 530.758,Z 536.239,A -85,B 0,C 180,E1 -4417.8,E2 -4417.8} C_VEL
LIN {X 0,Y 530.931,Z 527.994,A -85,B 0,C 180,E1 -4418.948,E2 -4418.948} C_VEL
LIN {X 0,Y 531.114,Z 519.542,A -85,B 0,C 180,E1 -4419.905,E2 -4419.905} C_VEL
LIN {X 0,Y 531.41,Z 509.103,A -85,B 0,C 180,E1 -4420.862,E2 -4420.862} C_VEL
LIN {X 0,Y 531.645,Z 498.393,A -85,B 0,C 180,E1 -4421.655,E2 -4421.655} C_VEL
LIN {X 0,Y 531.856,Z 487.418,A -85,B 0,C 180,E1 -4422.302,E2 -4422.302} C_VEL
LIN {X 0,Y 532.107,Z 475.776,A -85,B 0,C 180,E1 -4422.829,E2 -4422.829} C_VEL
LIN {X 0,Y 532.322,Z 462.365,A -85,B 0,C 180,E1 -4423.261,E2 -4423.261} C_VEL
LIN {X 0,Y 530.697,Z 451.532,A -85,B 0,C 180,E1 -4423.546,E2 -4423.546} C_VEL
LIN {X 0,Y 530.816,Z 442.761,A -85,B 0,C 180,E1 -4426.143,E2 -4426.143} C_VEL
LIN {X 0,Y 530.962,Z 433.494,A -85,B 0,C 180,E1 -4428.922,E2 -4428.922} C_VEL
LIN {X 0,Y 531.115,Z 424.227,A -85,B 0,C 180,E1 -4431.746,E2 -4431.746} C_VEL
LIN {X 0,Y 531.318,Z 414.96,A -85,B 0,C 180,E1 -4434.624,E2 -4434.624} C_VEL
LIN {X 0,Y 531.49,Z 405.499,A -85,B 0,C 180,E1 -4437.63,E2 -4437.63} C_VEL
LIN {X 0,Y 531.743,Z 395.804,A -85,B 0,C 180,E1 -4440.784,E2 -4440.784} C_VEL
LIN {X 0,Y 532.009,Z 387.005,A -85,B 0,C 180,E1 -4443.698,E2 -4443.698} C_VEL
LIN {X 0,Y 532.062,Z 380.532,A -85,B 0,C 180,E1 -4445.912,E2 -4445.912} C_VEL
LIN {X 0,Y 530.961,Z 374.35,A -85,B 0,C 180,E1 -4448.288,E2 -4448.288} C_VEL
LIN {X 0,Y 530.993,Z 374.344,A -85,B 0,C 180,E1 -4451.434,E2 -4451.434} C_VEL
LIN {X 0,Y 530.983,Z 374.345,A -85,B 0,C 180,E1 -4454.546,E2 -4454.546} C_VEL
LIN {X 0,Y 530.982,Z 374.345,A -85,B 0,C 180,E1 -4457.833,E2 -4457.833} C_VEL
LIN {X 0,Y 531,Z 374.345,A -85,B 0,C 180,E1 -4460.558,E2 -4460.558} C_VEL
LIN {X 0,Y 530.967,Z 374.348,A -85,B 0,C 180,E1 -4463.842,E2 -4463.842} C_VEL
LIN {X 0,Y 530.993,Z 374.345,A -85,B 0,C 180,E1 -4466.493,E2 -4466.493} C_VEL
LIN {X 0,Y 530.967,Z 374.349,A -85,B 0,C 180,E1 -4469.354,E2 -4469.354} C_VEL
LIN {X 0,Y 531.01,Z 374.342,A -85,B 0,C 180,E1 -4472.466,E2 -4472.466} C_VEL
LIN {X 0,Y 531,Z 374.345,A -85,B 0,C 180,E1 -4474.942,E2 -4474.942} C_VEL
LIN {X 0,Y 530.963,Z 374.348,A -85,B 0,C 180,E1 -4478.246,E2 -4478.246} C_VEL
LIN {X 0,Y 530.989,Z 374.346,A -85,B 0,C 180,E1 -4480.677,E2 -4480.677} C_VEL
LIN {X 0,Y 530.985,Z 374.345,A -85,B 0,C 180,E1 -4483.071,E2 -4483.071} C_VEL
LIN {X 0,Y 531.009,Z 374.341,A -85,B 0,C 180,E1 -4485.436,E2 -4485.436} C_VEL
LIN {X 0,Y 531.037,Z 374.34,A -85,B 0,C 180,E1 -4488.55,E2 -4488.55} C_VEL
LIN {X 0,Y 531.052,Z 374.337,A -85,B 0,C 180,E1 -4491.629,E2 -4491.629} C_VEL
LIN {X 0,Y 531.112,Z 374.33,A -85,B 0,C 180,E1 -4494.685,E2 -4494.685} C_VEL
LIN {X 0,Y 531.13,Z 374.325,A -85,B 0,C 180,E1 -4497.725,E2 -4497.725} C_VEL
LIN {X 0,Y 531.148,Z 374.325,A -85,B 0,C 180,E1 -4500.758,E2 -4500.758} C_VEL
LIN {X 0,Y 531.101,Z 374.33,A -85,B 0,C 180,E1 -4503.034,E2 -4503.034} C_VEL
LIN {X 0,Y 531.076,Z 374.335,A -85,B 0,C 180,E1 -4506.077,E2 -4506.077} C_VEL
LIN {X 0,Y 531.029,Z 374.341,A -85,B 0,C 180,E1 -4509.138,E2 -4509.138} C_VEL
LIN {X 0,Y 531.032,Z 374.339,A -85,B 0,C 180,E1 -4512.225,E2 -4512.225} C_VEL
LIN {X 0,Y 530.987,Z 374.343,A -85,B 0,C 180,E1 -4515.35,E2 -4515.35} C_VEL
LIN {X 0,Y 531.008,Z 374.341,A -85,B 0,C 180,E1 -4517.723,E2 -4517.723} C_VEL
LIN {X 0,Y 530.994,Z 374.343,A -85,B 0,C 180,E1 -4520.938,E2 -4520.938} C_VEL
LIN {X 0,Y 530.972,Z 374.347,A -85,B 0,C 180,E1 -4524.225,E2 -4524.225} C_VEL
LIN {X 0,Y 531.005,Z 374.343,A -85,B 0,C 180,E1 -4526.744,E2 -4526.744} C_VEL
LIN {X 0,Y 530.976,Z 374.347,A -85,B 0,C 180,E1 -4529.323,E2 -4529.323} C_VEL
LIN {X 0,Y 530.974,Z 374.346,A -85,B 0,C 180,E1 -4532.104,E2 -4532.104} C_VEL
LIN {X 0,Y 530.986,Z 374.345,A -85,B 0,C 180,E1 -4534.855,E2 -4534.855} C_VEL
LIN {X 0,Y 530.963,Z 374.347,A -85,B 0,C 180,E1 -4537.508,E2 -4537.508} C_VEL
LIN {X 0,Y 531.022,Z 374.342,A -85,B 0,C 180,E1 -4540.43,E2 -4540.43} C_VEL
LIN {X 0,Y 530.948,Z 374.349,A -85,B 0,C 180,E1 -4543.571,E2 -4543.571} C_VEL
LIN {X 0,Y 530.279,Z 374.433,A -85,B 0,C 180,E1 -4544.204,E2 -4544.204} C_VEL
LIN {X 0,Y 527.434,Z 374.788,A -85,B 0,C 180,E1 -4545.233,E2 -4545.233} C_VEL
LIN {X 0,Y 525.032,Z 375.09,A -85,B 0,C 180,E1 -4546.062,E2 -4546.062} C_VEL
LIN {X 0,Y 524,Z 375.217,A -85,B 0,C 180,E1 -4546.701,E2 -4546.701} C_VEL
LIN {X 0,Y 523.916,Z 375.226,A -85,B 0,C 180,E1 -4546.918,E2 -4546.918} C_VEL
LIN {X 0,Y 523.946,Z 375.222,A -85,B 0,C 180,E1 -4549.922,E2 -4549.922} C_VEL
LIN {X 0,Y 523.909,Z 375.225,A -85,B 0,C 180,E1 -4552.869,E2 -4552.869} C_VEL
LIN {X 0,Y 523.94,Z 375.223,A -85,B 0,C 180,E1 -4555.711,E2 -4555.711} C_VEL
LIN {X 0,Y 523.923,Z 375.224,A -85,B 0,C 180,E1 -4558.457,E2 -4558.457} C_VEL
LIN {X 0,Y 523.94,Z 375.222,A -85,B 0,C 180,E1 -4561.126,E2 -4561.126} C_VEL
LIN {X 0,Y 523.986,Z 375.217,A -85,B 0,C 180,E1 -4563.981,E2 -4563.981} C_VEL
LIN {X 0,Y 523.939,Z 375.223,A -85,B 0,C 180,E1 -4566.272,E2 -4566.272} C_VEL
LIN {X 0,Y 523.947,Z 375.221,A -85,B 0,C 180,E1 -4568.767,E2 -4568.767} C_VEL
LIN {X 0,Y 523.951,Z 375.221,A -85,B 0,C 180,E1 -4571.221,E2 -4571.221} C_VEL
LIN {X 0,Y 523.936,Z 375.225,A -85,B 0,C 180,E1 -4573.639,E2 -4573.639} C_VEL
LIN {X 0,Y 523.943,Z 375.223,A -85,B 0,C 180,E1 -4576.029,E2 -4576.029} C_VEL
LIN {X 0,Y 524.017,Z 375.212,A -85,B 0,C 180,E1 -4578.395,E2 -4578.395} C_VEL
LIN {X 0,Y 524.004,Z 375.216,A -85,B 0,C 180,E1 -4581.516,E2 -4581.516} C_VEL
LIN {X 0,Y 524.086,Z 375.205,A -85,B 0,C 180,E1 -4584.614,E2 -4584.614} C_VEL
LIN {X 0,Y 523.879,Z 375.234,A -85,B 0,C 180,E1 -4588.463,E2 -4588.463} C_VEL
LIN {X 0,Y 523.844,Z 375.245,A -85,B 0,C 180,E1 -4589.231,E2 -4589.231} C_VEL
LIN {X 0,Y 523.615,Z 377.8,A -85,B 0,C 180,E1 -4591.538,E2 -4591.538} C_VEL
LIN {X 0,Y 523.605,Z 381.224,A -85,B 0,C 180,E1 -4594.619,E2 -4594.619} C_VEL
LIN {X 0,Y 523.585,Z 383.803,A -85,B 0,C 180,E1 -4596.939,E2 -4596.939} C_VEL
LIN {X 0,Y 523.489,Z 387.292,A -85,B 0,C 180,E1 -4600.051,E2 -4600.051} C_VEL
LIN {X 0,Y 523.436,Z 389.866,A -85,B 0,C 180,E1 -4602.405,E2 -4602.405} C_VEL
LIN {X 0,Y 523.411,Z 393.392,A -85,B 0,C 180,E1 -4605.578,E2 -4605.578} C_VEL
LIN {X 0,Y 523.335,Z 396.572,A -85,B 0,C 180,E1 -4608.396,E2 -4608.396} C_VEL
LIN {X 0,Y 525.375,Z 407.341,A -85,B 0,C 180,E1 -4608.726,E2 -4608.726} C_VEL
LIN {X 0,Y 525.14,Z 419.965,A -85,B 0,C 180,E1 -4609.191,E2 -4609.191} C_VEL
LIN {X 0,Y 524.897,Z 431.331,A -85,B 0,C 180,E1 -4609.758,E2 -4609.758} C_VEL
LIN {X 0,Y 524.651,Z 442.65,A -85,B 0,C 180,E1 -4610.485,E2 -4610.485} C_VEL
LIN {X 0,Y 524.344,Z 452.957,A -85,B 0,C 180,E1 -4611.319,E2 -4611.319} C_VEL
LIN {X 0,Y 524.09,Z 462.649,A -85,B 0,C 180,E1 -4612.288,E2 -4612.288} C_VEL
LIN {X 0,Y 523.816,Z 471.052,A -85,B 0,C 180,E1 -4613.316,E2 -4613.316} C_VEL
LIN {X 0,Y 523.698,Z 477.788,A -85,B 0,C 180,E1 -4614.321,E2 -4614.321} C_VEL
LIN {X 0,Y 523.565,Z 483.933,A -85,B 0,C 180,E1 -4615.439,E2 -4615.439} C_VEL
LIN {X 0,Y 523.412,Z 489.522,A -85,B 0,C 180,E1 -4616.731,E2 -4616.731} C_VEL
LIN {X 0,Y 523.352,Z 493.747,A -85,B 0,C 180,E1 -4618.034,E2 -4618.034} C_VEL
LIN {X 0,Y 523.334,Z 496.456,A -85,B 0,C 180,E1 -4619.202,E2 -4619.202} C_VEL
LIN {X 0,Y 523.304,Z 498.592,A -85,B 0,C 180,E1 -4620.736,E2 -4620.736} C_VEL
LIN {X 0,Y 523.27,Z 499.139,A -85,B 0,C 180,E1 -4622.204,E2 -4622.204} C_VEL
LIN {X 0,Y 523.281,Z 498.319,A -85,B 0,C 180,E1 -4623.622,E2 -4623.622} C_VEL
LIN {X 0,Y 523.289,Z 496.274,A -85,B 0,C 180,E1 -4624.989,E2 -4624.989} C_VEL
LIN {X 0,Y 523.395,Z 493.012,A -85,B 0,C 180,E1 -4626.325,E2 -4626.325} C_VEL
LIN {X 0,Y 523.452,Z 488.552,A -85,B 0,C 180,E1 -4627.613,E2 -4627.613} C_VEL
LIN {X 0,Y 523.577,Z 482.815,A -85,B 0,C 180,E1 -4628.873,E2 -4628.873} C_VEL
LIN {X 0,Y 523.771,Z 475.68,A -85,B 0,C 180,E1 -4630.108,E2 -4630.108} C_VEL
LIN {X 0,Y 523.946,Z 466.933,A -85,B 0,C 180,E1 -4631.308,E2 -4631.308} C_VEL
LIN {X 0,Y 524.207,Z 458.006,A -85,B 0,C 180,E1 -4632.296,E2 -4632.296} C_VEL
LIN {X 0,Y 524.474,Z 447.418,A -85,B 0,C 180,E1 -4633.248,E2 -4633.248} C_VEL
LIN {X 0,Y 524.737,Z 437.215,A -85,B 0,C 180,E1 -4633.982,E2 -4633.982} C_VEL
LIN {X 0,Y 525.022,Z 425.95,A -85,B 0,C 180,E1 -4634.623,E2 -4634.623} C_VEL
LIN {X 0,Y 525.271,Z 413.431,A -85,B 0,C 180,E1 -4635.163,E2 -4635.163} C_VEL
LIN {X 0,Y 525.181,Z 406.62,A -85,B 0,C 180,E1 -4635.395,E2 -4635.395} C_VEL
LIN {X 0,Y 523.315,Z 396.695,A -85,B 0,C 180,E1 -4635.705,E2 -4635.705} C_VEL
LIN {X 0,Y 523.348,Z 393.225,A -85,B 0,C 180,E1 -4638.851,E2 -4638.851} C_VEL
LIN {X 0,Y 523.374,Z 389.984,A -85,B 0,C 180,E1 -4641.851,E2 -4641.851} C_VEL
LIN {X 0,Y 523.462,Z 386.847,A -85,B 0,C 180,E1 -4644.738,E2 -4644.738} C_VEL
LIN {X 0,Y 523.55,Z 383.579,A -85,B 0,C 180,E1 -4647.745,E2 -4647.745} C_VEL
LIN {X 0,Y 523.591,Z 380.892,A -85,B 0,C 180,E1 -4650.222,E2 -4650.222} C_VEL
LIN {X 0,Y 523.594,Z 378.057,A -85,B 0,C 180,E1 -4652.847,E2 -4652.847} C_VEL
LIN {X 0,Y 523.685,Z 375.257,A -85,B 0,C 180,E1 -4655.416,E2 -4655.416} C_VEL
LIN {X 0,Y 523.928,Z 375.225,A -85,B 0,C 180,E1 -4657.939,E2 -4657.939} C_VEL
LIN {X 0,Y 523.971,Z 375.219,A -85,B 0,C 180,E1 -4660.408,E2 -4660.408} C_VEL
LIN {X 0,Y 523.961,Z 375.219,A -85,B 0,C 180,E1 -4662.837,E2 -4662.837} C_VEL
LIN {X 0,Y 523.97,Z 375.218,A -85,B 0,C 180,E1 -4665.235,E2 -4665.235} C_VEL
LIN {X 0,Y 524.006,Z 375.215,A -85,B 0,C 180,E1 -4668.394,E2 -4668.394} C_VEL
LIN {X 0,Y 523.999,Z 375.215,A -85,B 0,C 180,E1 -4671.516,E2 -4671.516} C_VEL
LIN {X 0,Y 524.079,Z 375.204,A -85,B 0,C 180,E1 -4674.614,E2 -4674.614} C_VEL
LIN {X 0,Y 524.106,Z 375.201,A -85,B 0,C 180,E1 -4677.694,E2 -4677.694} C_VEL
LIN {X 0,Y 524.12,Z 375.2,A -85,B 0,C 180,E1 -4680.768,E2 -4680.768} C_VEL
LIN {X 0,Y 524.068,Z 375.206,A -85,B 0,C 180,E1 -4683.075,E2 -4683.075} C_VEL
LIN {X 0,Y 524.039,Z 375.21,A -85,B 0,C 180,E1 -4686.159,E2 -4686.159} C_VEL
LIN {X 0,Y 523.994,Z 375.215,A -85,B 0,C 180,E1 -4689.262,E2 -4689.262} C_VEL
LIN {X 0,Y 524.002,Z 375.214,A -85,B 0,C 180,E1 -4691.743,E2 -4691.743} C_VEL
LIN {X 0,Y 523.986,Z 375.217,A -85,B 0,C 180,E1 -4695.052,E2 -4695.052} C_VEL
LIN {X 0,Y 523.959,Z 375.219,A -85,B 0,C 180,E1 -4697.969,E2 -4697.969} C_VEL
LIN {X 0,Y 523.966,Z 375.218,A -85,B 0,C 180,E1 -4700.41,E2 -4700.41} C_VEL
LIN {X 0,Y 523.911,Z 375.226,A -85,B 0,C 180,E1 -4702.894,E2 -4702.894} C_VEL
LIN {X 0,Y 523.95,Z 375.221,A -85,B 0,C 180,E1 -4705.419,E2 -4705.419} C_VEL
LIN {X 0,Y 523.966,Z 375.22,A -85,B 0,C 180,E1 -4707.999,E2 -4707.999} C_VEL
LIN {X 0,Y 523.939,Z 375.223,A -85,B 0,C 180,E1 -4710.855,E2 -4710.855} C_VEL
LIN {X 0,Y 523.926,Z 375.225,A -85,B 0,C 180,E1 -4713.73,E2 -4713.73} C_VEL
LIN {X 0,Y 523.899,Z 375.23,A -85,B 0,C 180,E1 -4716.402,E2 -4716.402} C_VEL
LIN {X 0,Y 523.956,Z 375.223,A -85,B 0,C 180,E1 -4719.082,E2 -4719.082} C_VEL
LIN {X 0,Y 523.954,Z 375.22,A -85,B 0,C 180,E1 -4722.119,E2 -4722.119} C_VEL
LIN {X 0,Y 523.952,Z 375.223,A -85,B 0,C 180,E1 -4725.309,E2 -4725.309} C_VEL
LIN {X 0,Y 523.96,Z 375.224,A -85,B 0,C 180,E1 -4728.689,E2 -4728.689} C_VEL
LIN {X 0,Y 523.943,Z 375.281,A -85,B 0,C 180,E1 -4731.473,E2 -4731.473} C_VEL
LIN {X 0,Y 525.057,Z 381.513,A -85,B 0,C 180,E1 -4733.918,E2 -4733.918} C_VEL
LIN {X 0,Y 525.03,Z 387.667,A -85,B 0,C 180,E1 -4736.091,E2 -4736.091} C_VEL
LIN {X 0,Y 524.77,Z 396.473,A -85,B 0,C 180,E1 -4738.995,E2 -4738.995} C_VEL
LIN {X 0,Y 524.514,Z 406.11,A -85,B 0,C 180,E1 -4742.171,E2 -4742.171} C_VEL
LIN {X 0,Y 524.31,Z 414.959,A -85,B 0,C 180,E1 -4745.025,E2 -4745.025} C_VEL
LIN {X 0,Y 524.124,Z 424.226,A -85,B 0,C 180,E1 -4747.948,E2 -4747.948} C_VEL
LIN {X 0,Y 523.928,Z 433.493,A -85,B 0,C 180,E1 -4750.814,E2 -4750.814} C_VEL
LIN {X 0,Y 523.764,Z 442.76,A -85,B 0,C 180,E1 -4753.633,E2 -4753.633} C_VEL
LIN {X 0,Y 523.647,Z 451.736,A -85,B 0,C 180,E1 -4756.286,E2 -4756.286} C_VEL
LIN {X 0,Y 525.416,Z 463.271,A -85,B 0,C 180,E1 -4756.586,E2 -4756.586} C_VEL
LIN {X 0,Y 525.191,Z 475.772,A -85,B 0,C 180,E1 -4756.998,E2 -4756.998} C_VEL
LIN {X 0,Y 524.929,Z 487.411,A -85,B 0,C 180,E1 -4757.532,E2 -4757.532} C_VEL
LIN {X 0,Y 524.662,Z 498.824,A -85,B 0,C 180,E1 -4758.218,E2 -4758.218} C_VEL
LIN {X 0,Y 524.394,Z 510.262,A -85,B 0,C 180,E1 -4759.088,E2 -4759.088} C_VEL
LIN {X 0,Y 524.096,Z 519.539,A -85,B 0,C 180,E1 -4759.961,E2 -4759.961} C_VEL
LIN {X 0,Y 523.896,Z 527.991,A -85,B 0,C 180,E1 -4760.931,E2 -4760.931} C_VEL
LIN {X 0,Y 523.688,Z 536.237,A -85,B 0,C 180,E1 -4762.093,E2 -4762.093} C_VEL
LIN {X 0,Y 523.575,Z 541.868,A -85,B 0,C 180,E1 -4763.061,E2 -4763.061} C_VEL
LIN {X 0,Y 523.544,Z 547.366,A -85,B 0,C 180,E1 -4764.222,E2 -4764.222} C_VEL
LIN {X 0,Y 523.361,Z 551.677,A -85,B 0,C 180,E1 -4765.378,E2 -4765.378} C_VEL
LIN {X 0,Y 523.443,Z 553.957,A -85,B 0,C 180,E1 -4766.151,E2 -4766.151} C_VEL
LIN {X 0,Y 523.367,Z 555.808,A -85,B 0,C 180,E1 -4766.921,E2 -4766.921} C_VEL
LIN {X 0,Y 523.335,Z 557.197,A -85,B 0,C 180,E1 -4767.691,E2 -4767.691} C_VEL
LIN {X 0,Y 523.25,Z 558.785,A -85,B 0,C 180,E1 -4769.23,E2 -4769.23} C_VEL
LIN {X 0,Y 523.246,Z 559,A -85,B 0,C 180,E1 -4770,E2 -4770} C_VEL
LIN {X 0,Y 523.275,Z 558.186,A -85,B 0,C 180,E1 -4771.539,E2 -4771.539} C_VEL
LIN {X 0,Y 523.335,Z 557.199,A -85,B 0,C 180,E1 -4772.309,E2 -4772.309} C_VEL
LIN {X 0,Y 523.367,Z 555.81,A -85,B 0,C 180,E1 -4773.079,E2 -4773.079} C_VEL
LIN {X 0,Y 523.441,Z 552.896,A -85,B 0,C 180,E1 -4774.235,E2 -4774.235} C_VEL
LIN {X 0,Y 523.464,Z 548.95,A -85,B 0,C 180,E1 -4775.392,E2 -4775.392} C_VEL
LIN {X 0,Y 523.523,Z 543.728,A -85,B 0,C 180,E1 -4776.581,E2 -4776.581} C_VEL
LIN {X 0,Y 523.664,Z 537.47,A -85,B 0,C 180,E1 -4777.712,E2 -4777.712} C_VEL
LIN {X 0,Y 523.857,Z 529.481,A -85,B 0,C 180,E1 -4778.875,E2 -4778.875} C_VEL
LIN {X 0,Y 524.086,Z 521.339,A -85,B 0,C 180,E1 -4779.844,E2 -4779.844} C_VEL
LIN {X 0,Y 524.352,Z 511.405,A -85,B 0,C 180,E1 -4780.815,E2 -4780.815} C_VEL
LIN {X 0,Y 524.639,Z 500.205,A -85,B 0,C 180,E1 -4781.688,E2 -4781.688} C_VEL
LIN {X 0,Y 524.845,Z 489.184,A -85,B 0,C 180,E1 -4782.371,E2 -4782.371} C_VEL
LIN {X 0,Y 525.144,Z 476.989,A -85,B 0,C 180,E1 -4782.953,E2 -4782.953} C_VEL
LIN {X 0,Y 525.377,Z 464.193,A -85,B 0,C 180,E1 -4783.39,E2 -4783.39} C_VEL
LIN {X 0,Y 525.064,Z 460.302,A -85,B 0,C 180,E1 -4783.503,E2 -4783.503} C_VEL
LIN {X 0,Y 523.635,Z 451.532,A -85,B 0,C 180,E1 -4783.732,E2 -4783.732} C_VEL
LIN {X 0,Y 523.793,Z 441.437,A -85,B 0,C 180,E1 -4786.766,E2 -4786.766} C_VEL
LIN {X 0,Y 523.957,Z 432.17,A -85,B 0,C 180,E1 -4789.592,E2 -4789.592} C_VEL
LIN {X 0,Y 524.126,Z 423.44,A -85,B 0,C 180,E1 -4792.298,E2 -4792.298} C_VEL
LIN {X 0,Y 524.349,Z 413.636,A -85,B 0,C 180,E1 -4795.397,E2 -4795.397} C_VEL
LIN {X 0,Y 524.6,Z 404.369,A -85,B 0,C 180,E1 -4798.397,E2 -4798.397} C_VEL
LIN {X 0,Y 524.816,Z 394.992,A -85,B 0,C 180,E1 -4801.483,E2 -4801.483} C_VEL
LIN {X 0,Y 525.08,Z 386.931,A -85,B 0,C 180,E1 -4804.204,E2 -4804.204} C_VEL
LIN {X 0,Y 525.075,Z 381.547,A -85,B 0,C 180,E1 -4806.08,E2 -4806.08} C_VEL
LIN {X 0,Y 523.931,Z 375.225,A -85,B 0,C 180,E1 -4808.589,E2 -4808.589} C_VEL
LIN {X 0,Y 523.955,Z 375.221,A -85,B 0,C 180,E1 -4811.31,E2 -4811.31} C_VEL
LIN {X 0,Y 523.951,Z 375.221,A -85,B 0,C 180,E1 -4814.691,E2 -4814.691} C_VEL
LIN {X 0,Y 523.951,Z 375.221,A -85,B 0,C 180,E1 -4817.881,E2 -4817.881} C_VEL
LIN {X 0,Y 523.954,Z 375.222,A -85,B 0,C 180,E1 -4820.918,E2 -4820.918} C_VEL
LIN {X 0,Y 523.922,Z 375.225,A -85,B 0,C 180,E1 -4823.827,E2 -4823.827} C_VEL
LIN {X 0,Y 523.937,Z 375.223,A -85,B 0,C 180,E1 -4826.635,E2 -4826.635} C_VEL
LIN {X 0,Y 523.949,Z 375.223,A -85,B 0,C 180,E1 -4829.355,E2 -4829.355} C_VEL
LIN {X 0,Y 523.973,Z 375.218,A -85,B 0,C 180,E1 -4832.28,E2 -4832.28} C_VEL
LIN {X 0,Y 523.946,Z 375.222,A -85,B 0,C 180,E1 -4834.581,E2 -4834.581} C_VEL
LIN {X 0,Y 523.908,Z 375.228,A -85,B 0,C 180,E1 -4837.106,E2 -4837.106} C_VEL
LIN {X 0,Y 523.97,Z 375.218,A -85,B 0,C 180,E1 -4839.865,E2 -4839.865} C_VEL
LIN {X 0,Y 523.962,Z 375.222,A -85,B 0,C 180,E1 -4842.837,E2 -4842.837} C_VEL
LIN {X 0,Y 523.967,Z 375.219,A -85,B 0,C 180,E1 -4845.235,E2 -4845.235} C_VEL
LIN {X 0,Y 524.002,Z 375.217,A -85,B 0,C 180,E1 -4848.394,E2 -4848.394} C_VEL
LIN {X 0,Y 523.999,Z 375.216,A -85,B 0,C 180,E1 -4851.516,E2 -4851.516} C_VEL
LIN {X 0,Y 524.073,Z 375.206,A -85,B 0,C 180,E1 -4854.614,E2 -4854.614} C_VEL
LIN {X 0,Y 524.102,Z 375.201,A -85,B 0,C 180,E1 -4857.695,E2 -4857.695} C_VEL
LIN {X 0,Y 524.118,Z 375.201,A -85,B 0,C 180,E1 -4860.768,E2 -4860.768} C_VEL
LIN {X 0,Y 524.067,Z 375.206,A -85,B 0,C 180,E1 -4863.075,E2 -4863.075} C_VEL
LIN {X 0,Y 524.038,Z 375.212,A -85,B 0,C 180,E1 -4866.159,E2 -4866.159} C_VEL
LIN {X 0,Y 523.996,Z 375.216,A -85,B 0,C 180,E1 -4869.262,E2 -4869.262} C_VEL
LIN {X 0,Y 523.999,Z 375.216,A -85,B 0,C 180,E1 -4871.743,E2 -4871.743} C_VEL
LIN {X 0,Y 523.983,Z 375.217,A -85,B 0,C 180,E1 -4875.053,E2 -4875.053} C_VEL
LIN {X 0,Y 523.956,Z 375.22,A -85,B 0,C 180,E1 -4877.969,E2 -4877.969} C_VEL
LIN {X 0,Y 523.964,Z 375.222,A -85,B 0,C 180,E1 -4880.411,E2 -4880.411} C_VEL
LIN {X 0,Y 523.909,Z 375.226,A -85,B 0,C 180,E1 -4882.894,E2 -4882.894} C_VEL
LIN {X 0,Y 523.947,Z 375.22,A -85,B 0,C 180,E1 -4885.419,E2 -4885.419} C_VEL
LIN {X 0,Y 523.964,Z 375.22,A -85,B 0,C 180,E1 -4887.999,E2 -4887.999} C_VEL
LIN {X 0,Y 523.94,Z 375.222,A -85,B 0,C 180,E1 -4890.856,E2 -4890.856} C_VEL
LIN {X 0,Y 523.957,Z 375.222,A -85,B 0,C 180,E1 -4893.736,E2 -4893.736} C_VEL
LIN {X 0,Y 523.92,Z 375.225,A -85,B 0,C 180,E1 -4896.406,E2 -4896.406} C_VEL
LIN {X 0,Y 523.955,Z 375.221,A -85,B 0,C 180,E1 -4899.082,E2 -4899.082} C_VEL
LIN {X 0,Y 523.952,Z 375.221,A -85,B 0,C 180,E1 -4902.119,E2 -4902.119} C_VEL
LIN {X 0,Y 523.951,Z 375.22,A -85,B 0,C 180,E1 -4905.31,E2 -4905.31} C_VEL
LIN {X 0,Y 523.916,Z 375.226,A -85,B 0,C 180,E1 -4906.918,E2 -4906.918} C_VEL
LIN {X 0,Y 523.251,Z 375.308,A -85,B 0,C 180,E1 -4907.559,E2 -4907.559} C_VEL
LIN {X 0,Y 520.408,Z 375.665,A -85,B 0,C 180,E1 -4908.601,E2 -4908.601} C_VEL
LIN {X 0,Y 518.002,Z 375.968,A -85,B 0,C 180,E1 -4909.44,E2 -4909.44} C_VEL
LIN {X 0,Y 516.966,Z 376.095,A -85,B 0,C 180,E1 -4910.088,E2 -4910.088} C_VEL
LIN {X 0,Y 516.879,Z 376.104,A -85,B 0,C 180,E1 -4910.307,E2 -4910.307} C_VEL
LIN {X 0,Y 516.882,Z 376.101,A -85,B 0,C 180,E1 -4913.343,E2 -4913.343} C_VEL
LIN {X 0,Y 516.91,Z 376.099,A -85,B 0,C 180,E1 -4916.122,E2 -4916.122} C_VEL
LIN {X 0,Y 516.891,Z 376.101,A -85,B 0,C 180,E1 -4918.936,E2 -4918.936} C_VEL
LIN {X 0,Y 516.92,Z 376.098,A -85,B 0,C 180,E1 -4921.586,E2 -4921.586} C_VEL
LIN {X 0,Y 516.933,Z 376.095,A -85,B 0,C 180,E1 -4924.212,E2 -4924.212} C_VEL
LIN {X 0,Y 516.874,Z 376.103,A -85,B 0,C 180,E1 -4926.777,E2 -4926.777} C_VEL
LIN {X 0,Y 516.941,Z 376.094,A -85,B 0,C 180,E1 -4929.732,E2 -4929.732} C_VEL
LIN {X 0,Y 516.923,Z 376.096,A -85,B 0,C 180,E1 -4932.596,E2 -4932.596} C_VEL
LIN {X 0,Y 516.946,Z 376.093,A -85,B 0,C 180,E1 -4935.031,E2 -4935.031} C_VEL
LIN {X 0,Y 516.97,Z 376.091,A -85,B 0,C 180,E1 -4938.234,E2 -4938.234} C_VEL
LIN {X 0,Y 516.969,Z 376.093,A -85,B 0,C 180,E1 -4941.4,E2 -4941.4} C_VEL
LIN {X 0,Y 517.015,Z 376.086,A -85,B 0,C 180,E1 -4943.757,E2 -4943.757} C_VEL
LIN {X 0,Y 516.858,Z 376.104,A -85,B 0,C 180,E1 -4946.102,E2 -4946.102} C_VEL
LIN {X 0,Y 516.811,Z 376.115,A -85,B 0,C 180,E1 -4949.221,E2 -4949.221} C_VEL
LIN {X 0,Y 516.542,Z 378.5,A -85,B 0,C 180,E1 -4951.559,E2 -4951.559} C_VEL
LIN {X 0,Y 516.547,Z 381.943,A -85,B 0,C 180,E1 -4954.683,E2 -4954.683} C_VEL
LIN {X 0,Y 516.506,Z 384.531,A -85,B 0,C 180,E1 -4957.034,E2 -4957.034} C_VEL
LIN {X 0,Y 516.438,Z 388.057,A -85,B 0,C 180,E1 -4960.19,E2 -4960.19} C_VEL
LIN {X 0,Y 516.355,Z 390.691,A -85,B 0,C 180,E1 -4962.578,E2 -4962.578} C_VEL
LIN {X 0,Y 516.379,Z 393.424,A -85,B 0,C 180,E1 -4964.986,E2 -4964.986} C_VEL
LIN {X 0,Y 516.268,Z 396.985,A -85,B 0,C 180,E1 -4968.199,E2 -4968.199} C_VEL
LIN {X 0,Y 518.503,Z 408.528,A -85,B 0,C 180,E1 -4968.574,E2 -4968.574} C_VEL
LIN {X 0,Y 518.231,Z 420.985,A -85,B 0,C 180,E1 -4969.046,E2 -4969.046} C_VEL
LIN {X 0,Y 517.961,Z 432.271,A -85,B 0,C 180,E1 -4969.622,E2 -4969.622} C_VEL
LIN {X 0,Y 517.7,Z 443.62,A -85,B 0,C 180,E1 -4970.372,E2 -4970.372} C_VEL
LIN {X 0,Y 517.357,Z 454.799,A -85,B 0,C 180,E1 -4971.308,E2 -4971.308} C_VEL
LIN {X 0,Y 517.098,Z 463.072,A -85,B 0,C 180,E1 -4972.157,E2 -4972.157} C_VEL
LIN {X 0,Y 516.798,Z 471.686,A -85,B 0,C 180,E1 -4973.227,E2 -4973.227} C_VEL
LIN {X 0,Y 516.656,Z 478.722,A -85,B 0,C 180,E1 -4974.301,E2 -4974.301} C_VEL
LIN {X 0,Y 516.522,Z 484.498,A -85,B 0,C 180,E1 -4975.379,E2 -4975.379} C_VEL
LIN {X 0,Y 516.364,Z 490.049,A -85,B 0,C 180,E1 -4976.689,E2 -4976.689} C_VEL
LIN {X 0,Y 516.32,Z 493.625,A -85,B 0,C 180,E1 -4977.777,E2 -4977.777} C_VEL
LIN {X 0,Y 516.29,Z 495.381,A -85,B 0,C 180,E1 -4978.453,E2 -4978.453} C_VEL
LIN {X 0,Y 516.243,Z 497.304,A -85,B 0,C 180,E1 -4979.392,E2 -4979.392} C_VEL
LIN {X 0,Y 516.204,Z 498.548,A -85,B 0,C 180,E1 -4980.248,E2 -4980.248} C_VEL
